LIN {X 0,Y 395.833,Z 526.81,A -85,B 0,C 180,E1 10637.81,E2 10637.81} C_VEL
LIN {X 0,Y 395.52,Z 526.81,A -85,B 0,C 180,E1 10644.894,E2 10644.894} C_VEL
LIN {X 0,Y 395.41,Z 526.81,A -85,B 0,C 180,E1 10649.844,E2 10649.844} C_VEL
LIN {X 0,Y 395.216,Z 526.81,A -85,B 0,C 180,E1 10656.446,E2 10656.446} C_VEL
LIN {X 0,Y 395.064,Z 526.81,A -85,B 0,C 180,E1 10663.606,E2 10663.606} C_VEL
LIN {X 0,Y 395.094,Z 526.81,A -85,B 0,C 180,E1 10670.021,E2 10670.021} C_VEL
LIN {X 0,Y 395.236,Z 526.81,A -85,B 0,C 180,E1 10677.573,E2 10677.573} C_VEL
LIN {X 0,Y 395.461,Z 526.81,A -85,B 0,C 180,E1 10679.651,E2 10679.651} C_VEL
LIN {X 0,Y 410.092,Z 574.473,A -85,B 0,C 180,E1 10681.377,E2 10681.377} C_VEL
LIN {X 0,Y 408.745,Z 609.401,A -85,B 0,C 180,E1 10682.378,E2 10682.378} C_VEL
LIN {X 0,Y 406.158,Z 642.659,A -85,B 0,C 180,E1 10684.177,E2 10684.177} C_VEL
LIN {X 0,Y 403.313,Z 673.055,A -85,B 0,C 180,E1 10686.737,E2 10686.737} C_VEL
LIN {X 0,Y 400.568,Z 700.736,A -85,B 0,C 180,E1 10690.118,E2 10690.118} C_VEL
LIN {X 0,Y 398.689,Z 723.257,A -85,B 0,C 180,E1 10694.024,E2 10694.024} C_VEL
LIN {X 0,Y 397.841,Z 740.947,A -85,B 0,C 180,E1 10698.48,E2 10698.48} C_VEL
LIN {X 0,Y 397.641,Z 746.134,A -85,B 0,C 180,E1 10700.254,E2 10700.254} C_VEL
LIN {X 0,Y 395.186,Z 750.11,A -85,B 0,C 180,E1 10702.034,E2 10702.034} C_VEL
LIN {X 0,Y 390.021,Z 754.134,A -85,B 0,C 180,E1 10704.784,E2 10704.784} C_VEL
LIN {X 0,Y 389.948,Z 754.482,A -85,B 0,C 180,E1 10705.103,E2 10705.103} C_VEL
LIN {X 0,Y 390.043,Z 756.982,A -85,B 0,C 180,E1 10707.781,E2 10707.781} C_VEL
LIN {X 0,Y 390.037,Z 756.855,A -85,B 0,C 180,E1 10712.23,E2 10712.23} C_VEL
LIN {X 0,Y 389.934,Z 751.669,A -85,B 0,C 180,E1 10716.695,E2 10716.695} C_VEL
LIN {X 0,Y 389.895,Z 741.071,A -85,B 0,C 180,E1 10721.201,E2 10721.201} C_VEL
LIN {X 0,Y 390.787,Z 724.457,A -85,B 0,C 180,E1 10725.742,E2 10725.742} C_VEL
LIN {X 0,Y 392.693,Z 701.933,A -85,B 0,C 180,E1 10730.001,E2 10730.001} C_VEL
LIN {X 0,Y 395.677,Z 676.121,A -85,B 0,C 180,E1 10733.488,E2 10733.488} C_VEL
LIN {X 0,Y 399.365,Z 644.916,A -85,B 0,C 180,E1 10736.459,E2 10736.459} C_VEL
LIN {X 0,Y 402.863,Z 611.392,A -85,B 0,C 180,E1 10738.55,E2 10738.55} C_VEL
LIN {X 0,Y 405.252,Z 576.378,A -85,B 0,C 180,E1 10739.789,E2 10739.789} C_VEL
LIN {X 0,Y 399.916,Z 555.834,A -85,B 0,C 180,E1 10740.82,E2 10740.82} C_VEL
LIN {X 0,Y 389.16,Z 531.813,A -85,B 0,C 180,E1 10742.683,E2 10742.683} C_VEL
LIN {X 0,Y 387.296,Z 526.81,A -85,B 0,C 180,E1 10743.189,E2 10743.189} C_VEL
LIN {X 0,Y 387.265,Z 526.81,A -85,B 0,C 180,E1 10748.729,E2 10748.729} C_VEL
LIN {X 0,Y 387.23,Z 526.81,A -85,B 0,C 180,E1 10755.28,E2 10755.28} C_VEL
LIN {X 0,Y 387.272,Z 526.81,A -85,B 0,C 180,E1 10761.445,E2 10761.445} C_VEL
LIN {X 0,Y 387.353,Z 526.81,A -85,B 0,C 180,E1 10766.833,E2 10766.833} C_VEL
LIN {X 0,Y 387.496,Z 526.81,A -85,B 0,C 180,E1 10773.997,E2 10773.997} C_VEL
LIN {X 0,Y 387.667,Z 527.164,A -85,B 0,C 180,E1 10777.454,E2 10777.454} C_VEL
LIN {X 0,Y 397.662,Z 554.122,A -85,B 0,C 180,E1 10779.969,E2 10779.969} C_VEL
LIN {X 0,Y 400.192,Z 572.611,A -85,B 0,C 180,E1 10781.611,E2 10781.611} C_VEL
LIN {X 0,Y 397.581,Z 598.094,A -85,B 0,C 180,E1 10784.122,E2 10784.122} C_VEL
LIN {X 0,Y 395.193,Z 617.876,A -85,B 0,C 180,E1 10787.083,E2 10787.083} C_VEL
LIN {X 0,Y 393.153,Z 633.028,A -85,B 0,C 180,E1 10790.587,E2 10790.587} C_VEL
LIN {X 0,Y 391.819,Z 642.578,A -85,B 0,C 180,E1 10794.463,E2 10794.463} C_VEL
LIN {X 0,Y 391.065,Z 645.829,A -85,B 0,C 180,E1 10797.788,E2 10797.788} C_VEL
LIN {X 0,Y 390.664,Z 644.811,A -85,B 0,C 180,E1 10801.117,E2 10801.117} C_VEL
LIN {X 0,Y 390.812,Z 638.222,A -85,B 0,C 180,E1 10805.007,E2 10805.007} C_VEL
LIN {X 0,Y 391.409,Z 626.317,A -85,B 0,C 180,E1 10808.627,E2 10808.627} C_VEL
LIN {X 0,Y 392.534,Z 608.81,A -85,B 0,C 180,E1 10811.972,E2 10811.972} C_VEL
LIN {X 0,Y 393.989,Z 587.013,A -85,B 0,C 180,E1 10814.756,E2 10814.756} C_VEL
LIN {X 0,Y 395.236,Z 562.293,A -85,B 0,C 180,E1 10816.869,E2 10816.869} C_VEL
LIN {X 0,Y 389.321,Z 533.266,A -85,B 0,C 180,E1 10818.647,E2 10818.647} C_VEL
LIN {X 0,Y 388.01,Z 526.81,A -85,B 0,C 180,E1 10818.953,E2 10818.953} C_VEL
LIN {X 0,Y 387.53,Z 526.81,A -85,B 0,C 180,E1 10826.013,E2 10826.013} C_VEL
LIN {X 0,Y 387.291,Z 526.81,A -85,B 0,C 180,E1 10833.189,E2 10833.189} C_VEL
LIN {X 0,Y 387.238,Z 526.81,A -85,B 0,C 180,E1 10838.732,E2 10838.732} C_VEL
LIN {X 0,Y 387.183,Z 526.81,A -85,B 0,C 180,E1 10845.253,E2 10845.253} C_VEL
LIN {X 0,Y 387.29,Z 526.81,A -85,B 0,C 180,E1 10851.44,E2 10851.44} C_VEL
LIN {X 0,Y 387.348,Z 526.81,A -85,B 0,C 180,E1 10856.816,E2 10856.816} C_VEL
LIN {X 0,Y 387.543,Z 526.81,A -85,B 0,C 180,E1 10863.981,E2 10863.981} C_VEL
LIN {X 0,Y 387.824,Z 526.81,A -85,B 0,C 180,E1 10869.559,E2 10869.559} C_VEL
LIN {X 0,Y 387.949,Z 526.81,A -85,B 0,C 180,E1 10876.452,E2 10876.452} C_VEL
LIN {X 0,Y 388.374,Z 526.81,A -85,B 0,C 180,E1 10883.278,E2 10883.278} C_VEL
LIN {X 0,Y 388.755,Z 526.81,A -85,B 0,C 180,E1 10889.995,E2 10889.995} C_VEL
LIN {X 0,Y 388.368,Z 526.81,A -85,B 0,C 180,E1 10896.711,E2 10896.711} C_VEL
LIN {X 0,Y 388.065,Z 526.81,A -85,B 0,C 180,E1 10903.533,E2 10903.533} C_VEL
LIN {X 0,Y 387.816,Z 526.81,A -85,B 0,C 180,E1 10910.565,E2 10910.565} C_VEL
LIN {X 0,Y 387.507,Z 526.81,A -85,B 0,C 180,E1 10917.955,E2 10917.955} C_VEL
LIN {X 0,Y 387.3,Z 526.81,A -85,B 0,C 180,E1 10924.812,E2 10924.812} C_VEL
LIN {X 0,Y 387.148,Z 526.81,A -85,B 0,C 180,E1 10932.001,E2 10932.001} C_VEL
LIN {X 0,Y 387.205,Z 526.81,A -85,B 0,C 180,E1 10938.331,E2 10938.331} C_VEL
LIN {X 0,Y 387.318,Z 526.81,A -85,B 0,C 180,E1 10945.167,E2 10945.167} C_VEL
LIN {X 0,Y 387.523,Z 526.81,A -85,B 0,C 180,E1 10952.034,E2 10952.034} C_VEL
LIN {X 0,Y 387.831,Z 526.81,A -85,B 0,C 180,E1 10959.529,E2 10959.529} C_VEL
LIN {X 0,Y 387.974,Z 526.81,A -85,B 0,C 180,E1 10966.452,E2 10966.452} C_VEL
LIN {X 0,Y 388.422,Z 526.81,A -85,B 0,C 180,E1 10973.278,E2 10973.278} C_VEL
LIN {X 0,Y 388.722,Z 526.81,A -85,B 0,C 180,E1 10979.993,E2 10979.993} C_VEL
LIN {X 0,Y 388.356,Z 526.81,A -85,B 0,C 180,E1 10986.709,E2 10986.709} C_VEL
LIN {X 0,Y 388.004,Z 526.81,A -85,B 0,C 180,E1 10993.533,E2 10993.533} C_VEL
LIN {X 0,Y 387.766,Z 526.81,A -85,B 0,C 180,E1 11000.565,E2 11000.565} C_VEL
LIN {X 0,Y 387.519,Z 526.81,A -85,B 0,C 180,E1 11007.95,E2 11007.95} C_VEL
LIN {X 0,Y 387.354,Z 526.81,A -85,B 0,C 180,E1 11014.841,E2 11014.841} C_VEL
LIN {X 0,Y 387.099,Z 526.81,A -85,B 0,C 180,E1 11022.007,E2 11022.007} C_VEL
LIN {X 0,Y 387.065,Z 526.81,A -85,B 0,C 180,E1 11028.326,E2 11028.326} C_VEL
LIN {X 0,Y 387.244,Z 526.81,A -85,B 0,C 180,E1 11035.176,E2 11035.176} C_VEL
LIN {X 0,Y 387.526,Z 527.326,A -85,B 0,C 180,E1 11039.247,E2 11039.247} C_VEL
LIN {X 0,Y 402.597,Z 575.135,A -85,B 0,C 180,E1 11041.032,E2 11041.032} C_VEL
LIN {X 0,Y 401.08,Z 610.921,A -85,B 0,C 180,E1 11042.117,E2 11042.117} C_VEL
LIN {X 0,Y 398.473,Z 643.198,A -85,B 0,C 180,E1 11043.944,E2 11043.944} C_VEL
LIN {X 0,Y 395.477,Z 673.867,A -85,B 0,C 180,E1 11046.625,E2 11046.625} C_VEL
LIN {X 0,Y 392.717,Z 700.654,A -85,B 0,C 180,E1 11050.008,E2 11050.008} C_VEL
LIN {X 0,Y 390.815,Z 722.905,A -85,B 0,C 180,E1 11053.982,E2 11053.982} C_VEL
LIN {X 0,Y 389.989,Z 739.481,A -85,B 0,C 180,E1 11058.245,E2 11058.245} C_VEL
LIN {X 0,Y 389.898,Z 750.617,A -85,B 0,C 180,E1 11062.621,E2 11062.621} C_VEL
LIN {X 0,Y 389.948,Z 754.482,A -85,B 0,C 180,E1 11065.103,E2 11065.103} C_VEL
LIN {X 0,Y 387.658,Z 756.165,A -85,B 0,C 180,E1 11066.987,E2 11066.987} C_VEL
LIN {X 0,Y 382.341,Z 756.336,A -85,B 0,C 180,E1 11070.182,E2 11070.182} C_VEL
LIN {X 0,Y 382.162,Z 753.806,A -85,B 0,C 180,E1 11074.55,E2 11074.55} C_VEL
LIN {X 0,Y 381.944,Z 745.92,A -85,B 0,C 180,E1 11079.129,E2 11079.129} C_VEL
LIN {X 0,Y 382.319,Z 732.498,A -85,B 0,C 180,E1 11083.751,E2 11083.751} C_VEL
LIN {X 0,Y 383.876,Z 712.313,A -85,B 0,C 180,E1 11088.399,E2 11088.399} C_VEL
LIN {X 0,Y 386.838,Z 687.296,A -85,B 0,C 180,E1 11092.439,E2 11092.439} C_VEL
LIN {X 0,Y 390.458,Z 658.719,A -85,B 0,C 180,E1 11095.716,E2 11095.716} C_VEL
LIN {X 0,Y 394.404,Z 626.331,A -85,B 0,C 180,E1 11098.253,E2 11098.253} C_VEL
LIN {X 0,Y 397.556,Z 592.247,A -85,B 0,C 180,E1 11099.916,E2 11099.916} C_VEL
LIN {X 0,Y 398.025,Z 574.069,A -85,B 0,C 180,E1 11100.508,E2 11100.508} C_VEL
LIN {X 0,Y 390.505,Z 550.725,A -85,B 0,C 180,E1 11101.947,E2 11101.947} C_VEL
LIN {X 0,Y 379.376,Z 526.81,A -85,B 0,C 180,E1 11104.174,E2 11104.174} C_VEL
LIN {X 0,Y 379.266,Z 526.81,A -85,B 0,C 180,E1 11110.682,E2 11110.682} C_VEL
LIN {X 0,Y 379.263,Z 526.81,A -85,B 0,C 180,E1 11117.273,E2 11117.273} C_VEL
LIN {X 0,Y 379.297,Z 526.81,A -85,B 0,C 180,E1 11123.229,E2 11123.229} C_VEL
LIN {X 0,Y 379.446,Z 526.81,A -85,B 0,C 180,E1 11128.763,E2 11128.763} C_VEL
LIN {X 0,Y 379.632,Z 526.81,A -85,B 0,C 180,E1 11136.364,E2 11136.364} C_VEL
LIN {X 0,Y 390.489,Z 554.777,A -85,B 0,C 180,E1 11139.28,E2 11139.28} C_VEL
LIN {X 0,Y 393.345,Z 573.867,A -85,B 0,C 180,E1 11141.074,E2 11141.074} C_VEL
LIN {X 0,Y 390.46,Z 599.555,A -85,B 0,C 180,E1 11143.68,E2 11143.68} C_VEL
LIN {X 0,Y 387.805,Z 619.699,A -85,B 0,C 180,E1 11146.776,E2 11146.776} C_VEL
LIN {X 0,Y 385.589,Z 634.811,A -85,B 0,C 180,E1 11150.401,E2 11150.401} C_VEL
LIN {X 0,Y 384.111,Z 644.058,A -85,B 0,C 180,E1 11154.352,E2 11154.352} C_VEL
LIN {X 0,Y 383.311,Z 647.144,A -85,B 0,C 180,E1 11157.743,E2 11157.743} C_VEL
LIN {X 0,Y 382.849,Z 645.949,A -85,B 0,C 180,E1 11161.14,E2 11161.14} C_VEL
LIN {X 0,Y 383.023,Z 639.115,A -85,B 0,C 180,E1 11165.109,E2 11165.109} C_VEL
LIN {X 0,Y 383.623,Z 626.948,A -85,B 0,C 180,E1 11168.804,E2 11168.804} C_VEL
LIN {X 0,Y 384.818,Z 609.109,A -85,B 0,C 180,E1 11172.216,E2 11172.216} C_VEL
LIN {X 0,Y 386.298,Z 586.882,A -85,B 0,C 180,E1 11175.056,E2 11175.056} C_VEL
LIN {X 0,Y 387.223,Z 561.791,A -85,B 0,C 180,E1 11177.213,E2 11177.213} C_VEL
LIN {X 0,Y 381.165,Z 532.299,A -85,B 0,C 180,E1 11179.02,E2 11179.02} C_VEL
LIN {X 0,Y 380.043,Z 526.81,A -85,B 0,C 180,E1 11179.299,E2 11179.299} C_VEL
LIN {X 0,Y 379.646,Z 526.81,A -85,B 0,C 180,E1 11186.027,E2 11186.027} C_VEL
LIN {X 0,Y 379.396,Z 526.81,A -85,B 0,C 180,E1 11193.055,E2 11193.055} C_VEL
LIN {X 0,Y 379.195,Z 526.81,A -85,B 0,C 180,E1 11200.647,E2 11200.647} C_VEL
LIN {X 0,Y 379.23,Z 526.81,A -85,B 0,C 180,E1 11207.249,E2 11207.249} C_VEL
LIN {X 0,Y 379.307,Z 526.81,A -85,B 0,C 180,E1 11213.213,E2 11213.213} C_VEL
LIN {X 0,Y 379.447,Z 526.81,A -85,B 0,C 180,E1 11218.747,E2 11218.747} C_VEL
LIN {X 0,Y 379.66,Z 526.81,A -85,B 0,C 180,E1 11223.975,E2 11223.975} C_VEL
LIN {X 0,Y 379.934,Z 526.81,A -85,B 0,C 180,E1 11231.404,E2 11231.404} C_VEL
LIN {X 0,Y 380.094,Z 526.81,A -85,B 0,C 180,E1 11238.506,E2 11238.506} C_VEL
LIN {X 0,Y 380.536,Z 526.81,A -85,B 0,C 180,E1 11245.43,E2 11245.43} C_VEL
LIN {X 0,Y 380.853,Z 526.81,A -85,B 0,C 180,E1 11249.995,E2 11249.995} C_VEL
LIN {X 0,Y 380.457,Z 526.81,A -85,B 0,C 180,E1 11256.851,E2 11256.851} C_VEL
LIN {X 0,Y 380.121,Z 526.81,A -85,B 0,C 180,E1 11263.821,E2 11263.821} C_VEL
LIN {X 0,Y 379.834,Z 526.81,A -85,B 0,C 180,E1 11271.018,E2 11271.018} C_VEL
LIN {X 0,Y 379.524,Z 526.81,A -85,B 0,C 180,E1 11278.629,E2 11278.629} C_VEL
LIN {X 0,Y 379.366,Z 526.81,A -85,B 0,C 180,E1 11283.963,E2 11283.963} C_VEL
LIN {X 0,Y 379.166,Z 526.81,A -85,B 0,C 180,E1 11290.643,E2 11290.643} C_VEL
LIN {X 0,Y 379.233,Z 526.81,A -85,B 0,C 180,E1 11297.25,E2 11297.25} C_VEL
LIN {X 0,Y 379.283,Z 526.81,A -85,B 0,C 180,E1 11303.21,E2 11303.21} C_VEL
LIN {X 0,Y 379.42,Z 526.81,A -85,B 0,C 180,E1 11308.744,E2 11308.744} C_VEL
LIN {X 0,Y 379.709,Z 526.81,A -85,B 0,C 180,E1 11316.494,E2 11316.494} C_VEL
LIN {X 0,Y 379.995,Z 526.81,A -85,B 0,C 180,E1 11323.798,E2 11323.798} C_VEL
LIN {X 0,Y 380.291,Z 526.81,A -85,B 0,C 180,E1 11331.518,E2 11331.518} C_VEL
LIN {X 0,Y 380.78,Z 526.81,A -85,B 0,C 180,E1 11337.714,E2 11337.714} C_VEL
LIN {X 0,Y 380.594,Z 526.81,A -85,B 0,C 180,E1 11344.556,E2 11344.556} C_VEL
LIN {X 0,Y 380.149,Z 526.81,A -85,B 0,C 180,E1 11351.479,E2 11351.479} C_VEL
LIN {X 0,Y 379.929,Z 526.81,A -85,B 0,C 180,E1 11358.583,E2 11358.583} C_VEL
LIN {X 0,Y 379.626,Z 526.81,A -85,B 0,C 180,E1 11366.013,E2 11366.013} C_VEL
LIN {X 0,Y 379.446,Z 526.81,A -85,B 0,C 180,E1 11373.951,E2 11373.951} C_VEL
LIN {X 0,Y 379.154,Z 526.81,A -85,B 0,C 180,E1 11380.657,E2 11380.657} C_VEL
LIN {X 0,Y 379.074,Z 526.81,A -85,B 0,C 180,E1 11387.242,E2 11387.242} C_VEL
LIN {X 0,Y 379.181,Z 526.81,A -85,B 0,C 180,E1 11393.212,E2 11393.212} C_VEL
LIN {X 0,Y 379.575,Z 526.81,A -85,B 0,C 180,E1 11398.771,E2 11398.771} C_VEL
LIN {X 0,Y 395.009,Z 576.235,A -85,B 0,C 180,E1 11400.686,E2 11400.686} C_VEL
LIN {X 0,Y 393.505,Z 611.185,A -85,B 0,C 180,E1 11401.801,E2 11401.801} C_VEL
LIN {X 0,Y 390.686,Z 644.506,A -85,B 0,C 180,E1 11403.765,E2 11403.765} C_VEL
LIN {X 0,Y 387.684,Z 673.91,A -85,B 0,C 180,E1 11406.434,E2 11406.434} C_VEL
LIN {X 0,Y 384.8,Z 701.173,A -85,B 0,C 180,E1 11410.003,E2 11410.003} C_VEL
LIN {X 0,Y 382.933,Z 722.47,A -85,B 0,C 180,E1 11413.938,E2 11413.938} C_VEL
LIN {X 0,Y 382.09,Z 739.805,A -85,B 0,C 180,E1 11418.578,E2 11418.578} C_VEL
LIN {X 0,Y 382.104,Z 750.549,A -85,B 0,C 180,E1 11423.178,E2 11423.178} C_VEL
LIN {X 0,Y 382.217,Z 755.777,A -85,B 0,C 180,E1 11427.735,E2 11427.735} C_VEL
LIN {X 0,Y 382.341,Z 756.336,A -85,B 0,C 180,E1 11430.182,E2 11430.182} C_VEL
LIN {X 0,Y 379.656,Z 755.445,A -85,B 0,C 180,E1 11432.103,E2 11432.103} C_VEL
LIN {X 0,Y 374.266,Z 751.83,A -85,B 0,C 180,E1 11435.303,E2 11435.303} C_VEL
LIN {X 0,Y 374.054,Z 743.465,A -85,B 0,C 180,E1 11439.911,E2 11439.911} C_VEL
LIN {X 0,Y 374.633,Z 729.252,A -85,B 0,C 180,E1 11444.637,E2 11444.637} C_VEL
LIN {X 0,Y 376.399,Z 709.724,A -85,B 0,C 180,E1 11449.092,E2 11449.092} C_VEL
LIN {X 0,Y 379.627,Z 684.333,A -85,B 0,C 180,E1 11453.2,E2 11453.2} C_VEL
LIN {X 0,Y 383.506,Z 655.208,A -85,B 0,C 180,E1 11456.533,E2 11456.533} C_VEL
LIN {X 0,Y 387.98,Z 621.858,A -85,B 0,C 180,E1 11459.087,E2 11459.087} C_VEL
LIN {X 0,Y 391.317,Z 587.429,A -85,B 0,C 180,E1 11460.699,E2 11460.699} C_VEL
LIN {X 0,Y 391.301,Z 575.135,A -85,B 0,C 180,E1 11461.139,E2 11461.139} C_VEL
LIN {X 0,Y 383.806,Z 552.489,A -85,B 0,C 180,E1 11462.667,E2 11462.667} C_VEL
LIN {X 0,Y 372.915,Z 531.315,A -85,B 0,C 180,E1 11464.919,E2 11464.919} C_VEL
LIN {X 0,Y 371.481,Z 526.81,A -85,B 0,C 180,E1 11465.414,E2 11465.414} C_VEL
LIN {X 0,Y 371.381,Z 526.81,A -85,B 0,C 180,E1 11472.805,E2 11472.805} C_VEL
LIN {X 0,Y 371.368,Z 526.81,A -85,B 0,C 180,E1 11479.295,E2 11479.295} C_VEL
LIN {X 0,Y 371.392,Z 526.81,A -85,B 0,C 180,E1 11485.209,E2 11485.209} C_VEL
LIN {X 0,Y 371.555,Z 526.81,A -85,B 0,C 180,E1 11490.735,E2 11490.735} C_VEL
LIN {X 0,Y 371.721,Z 527.201,A -85,B 0,C 180,E1 11495.261,E2 11495.261} C_VEL
LIN {X 0,Y 383.001,Z 554.104,A -85,B 0,C 180,E1 11498.393,E2 11498.393} C_VEL
LIN {X 0,Y 386.609,Z 574.886,A -85,B 0,C 180,E1 11500.487,E2 11500.487} C_VEL
LIN {X 0,Y 383.394,Z 601.235,A -85,B 0,C 180,E1 11503.223,E2 11503.223} C_VEL
LIN {X 0,Y 380.485,Z 621.376,A -85,B 0,C 180,E1 11506.414,E2 11506.414} C_VEL
LIN {X 0,Y 378.267,Z 635.03,A -85,B 0,C 180,E1 11509.704,E2 11509.704} C_VEL
LIN {X 0,Y 376.74,Z 643.717,A -85,B 0,C 180,E1 11513.083,E2 11513.083} C_VEL
LIN {X 0,Y 376.091,Z 647.017,A -85,B 0,C 180,E1 11515.389,E2 11515.389} C_VEL
LIN {X 0,Y 375.545,Z 648.445,A -85,B 0,C 180,E1 11517.697,E2 11517.697} C_VEL
LIN {X 0,Y 375.051,Z 647.071,A -85,B 0,C 180,E1 11521.164,E2 11521.164} C_VEL
LIN {X 0,Y 375.204,Z 639.959,A -85,B 0,C 180,E1 11525.216,E2 11525.216} C_VEL
LIN {X 0,Y 375.844,Z 627.545,A -85,B 0,C 180,E1 11528.984,E2 11528.984} C_VEL
LIN {X 0,Y 377.082,Z 609.407,A -85,B 0,C 180,E1 11532.47,E2 11532.47} C_VEL
LIN {X 0,Y 378.751,Z 585.397,A -85,B 0,C 180,E1 11535.512,E2 11535.512} C_VEL
LIN {X 0,Y 379.458,Z 562.632,A -85,B 0,C 180,E1 11537.466,E2 11537.466} C_VEL
LIN {X 0,Y 373.527,Z 533.469,A -85,B 0,C 180,E1 11539.309,E2 11539.309} C_VEL
LIN {X 0,Y 372.132,Z 526.81,A -85,B 0,C 180,E1 11539.606,E2 11539.606} C_VEL
LIN {X 0,Y 371.66,Z 526.81,A -85,B 0,C 180,E1 11546.63,E2 11546.63} C_VEL
LIN {X 0,Y 371.482,Z 526.81,A -85,B 0,C 180,E1 11552.002,E2 11552.002} C_VEL
LIN {X 0,Y 371.281,Z 526.81,A -85,B 0,C 180,E1 11559.203,E2 11559.203} C_VEL
LIN {X 0,Y 371.309,Z 526.81,A -85,B 0,C 180,E1 11566.108,E2 11566.108} C_VEL
LIN {X 0,Y 371.306,Z 526.81,A -85,B 0,C 180,E1 11572.284,E2 11572.284} C_VEL
LIN {X 0,Y 371.539,Z 526.81,A -85,B 0,C 180,E1 11578.855,E2 11578.855} C_VEL
LIN {X 0,Y 371.751,Z 526.81,A -85,B 0,C 180,E1 11585.96,E2 11585.96} C_VEL
LIN {X 0,Y 371.967,Z 526.81,A -85,B 0,C 180,E1 11590.99,E2 11590.99} C_VEL
LIN {X 0,Y 372.154,Z 526.81,A -85,B 0,C 180,E1 11598.257,E2 11598.257} C_VEL
LIN {X 0,Y 372.623,Z 526.81,A -85,B 0,C 180,E1 11605.333,E2 11605.333} C_VEL
LIN {X 0,Y 372.951,Z 526.81,A -85,B 0,C 180,E1 11609.994,E2 11609.994} C_VEL
LIN {X 0,Y 372.53,Z 526.81,A -85,B 0,C 180,E1 11616.998,E2 11616.998} C_VEL
LIN {X 0,Y 372.178,Z 526.81,A -85,B 0,C 180,E1 11624.122,E2 11624.122} C_VEL
LIN {X 0,Y 371.857,Z 526.81,A -85,B 0,C 180,E1 11631.491,E2 11631.491} C_VEL
LIN {X 0,Y 371.632,Z 526.81,A -85,B 0,C 180,E1 11636.619,E2 11636.619} C_VEL
LIN {X 0,Y 371.484,Z 526.81,A -85,B 0,C 180,E1 11641.988,E2 11641.988} C_VEL
LIN {X 0,Y 371.252,Z 526.81,A -85,B 0,C 180,E1 11649.199,E2 11649.199} C_VEL
LIN {X 0,Y 371.291,Z 526.81,A -85,B 0,C 180,E1 11656.106,E2 11656.106} C_VEL
LIN {X 0,Y 371.286,Z 526.81,A -85,B 0,C 180,E1 11662.282,E2 11662.282} C_VEL
LIN {X 0,Y 371.509,Z 526.81,A -85,B 0,C 180,E1 11668.842,E2 11668.842} C_VEL
LIN {X 0,Y 371.732,Z 526.81,A -85,B 0,C 180,E1 11675.958,E2 11675.958} C_VEL
LIN {X 0,Y 371.991,Z 526.81,A -85,B 0,C 180,E1 11680.991,E2 11680.991} C_VEL
LIN {X 0,Y 372.17,Z 526.81,A -85,B 0,C 180,E1 11688.257,E2 11688.257} C_VEL
LIN {X 0,Y 372.61,Z 526.81,A -85,B 0,C 180,E1 11695.332,E2 11695.332} C_VEL
LIN {X 0,Y 372.837,Z 526.81,A -85,B 0,C 180,E1 11702.32,E2 11702.32} C_VEL
LIN {X 0,Y 372.351,Z 526.81,A -85,B 0,C 180,E1 11709.353,E2 11709.353} C_VEL
LIN {X 0,Y 372.084,Z 526.81,A -85,B 0,C 180,E1 11716.541,E2 11716.541} C_VEL
LIN {X 0,Y 371.814,Z 526.81,A -85,B 0,C 180,E1 11721.49,E2 11721.49} C_VEL
LIN {X 0,Y 371.654,Z 526.81,A -85,B 0,C 180,E1 11726.614,E2 11726.614} C_VEL
LIN {X 0,Y 371.508,Z 526.81,A -85,B 0,C 180,E1 11731.982,E2 11731.982} C_VEL
LIN {X 0,Y 371.276,Z 526.81,A -85,B 0,C 180,E1 11739.22,E2 11739.22} C_VEL
LIN {X 0,Y 371.162,Z 526.81,A -85,B 0,C 180,E1 11746.102,E2 11746.102} C_VEL
LIN {X 0,Y 371.173,Z 526.81,A -85,B 0,C 180,E1 11752.282,E2 11752.282} C_VEL
LIN {X 0,Y 371.62,Z 526.81,A -85,B 0,C 180,E1 11758.357,E2 11758.357} C_VEL
LIN {X 0,Y 387.541,Z 577.763,A -85,B 0,C 180,E1 11760.356,E2 11760.356} C_VEL
LIN {X 0,Y 385.852,Z 612.406,A -85,B 0,C 180,E1 11761.526,E2 11761.526} C_VEL
LIN {X 0,Y 382.941,Z 645.126,A -85,B 0,C 180,E1 11763.54,E2 11763.54} C_VEL
LIN {X 0,Y 379.793,Z 675.058,A -85,B 0,C 180,E1 11766.372,E2 11766.372} C_VEL
LIN {X 0,Y 376.896,Z 701.419,A -85,B 0,C 180,E1 11769.962,E2 11769.962} C_VEL
LIN {X 0,Y 374.984,Z 723.271,A -85,B 0,C 180,E1 11774.191,E2 11774.191} C_VEL
LIN {X 0,Y 374.23,Z 739.943,A -85,B 0,C 180,E1 11778.926,E2 11778.926} C_VEL
LIN {X 0,Y 374.273,Z 749.206,A -85,B 0,C 180,E1 11783.035,E2 11783.035} C_VEL
LIN {X 0,Y 374.409,Z 754.542,A -85,B 0,C 180,E1 11787.688,E2 11787.688} C_VEL
LIN {X 0,Y 374.401,Z 754.554,A -85,B 0,C 180,E1 11792.323,E2 11792.323} C_VEL
LIN {X 0,Y 374.266,Z 751.83,A -85,B 0,C 180,E1 11795.303,E2 11795.303} C_VEL
LIN {X 0,Y 371.643,Z 748.735,A -85,B 0,C 180,E1 11797.222,E2 11797.222} C_VEL
LIN {X 0,Y 366.27,Z 742.551,A -85,B 0,C 180,E1 11800.045,E2 11800.045} C_VEL
LIN {X 0,Y 366.196,Z 741.78,A -85,B 0,C 180,E1 11800.37,E2 11800.37} C_VEL
LIN {X 0,Y 366.888,Z 727.12,A -85,B 0,C 180,E1 11805.259,E2 11805.259} C_VEL
LIN {X 0,Y 368.886,Z 707.269,A -85,B 0,C 180,E1 11809.798,E2 11809.798} C_VEL
LIN {X 0,Y 372.458,Z 681.39,A -85,B 0,C 180,E1 11813.992,E2 11813.992} C_VEL
LIN {X 0,Y 376.746,Z 652.603,A -85,B 0,C 180,E1 11817.283,E2 11817.283} C_VEL
LIN {X 0,Y 381.426,Z 619.331,A -85,B 0,C 180,E1 11819.836,E2 11819.836} C_VEL
LIN {X 0,Y 384.969,Z 584.686,A -85,B 0,C 180,E1 11821.451,E2 11821.451} C_VEL
LIN {X 0,Y 384.345,Z 574.581,A -85,B 0,C 180,E1 11821.901,E2 11821.901} C_VEL
LIN {X 0,Y 375.655,Z 550.859,A -85,B 0,C 180,E1 11823.775,E2 11823.775} C_VEL
LIN {X 0,Y 365.632,Z 532.243,A -85,B 0,C 180,E1 11826.087,E2 11826.087} C_VEL
LIN {X 0,Y 363.398,Z 526.81,A -85,B 0,C 180,E1 11826.887,E2 11826.887} C_VEL
LIN {X 0,Y 363.432,Z 526.81,A -85,B 0,C 180,E1 11831.81,E2 11831.81} C_VEL
LIN {X 0,Y 363.426,Z 526.81,A -85,B 0,C 180,E1 11838.59,E2 11838.59} C_VEL
LIN {X 0,Y 363.414,Z 526.81,A -85,B 0,C 180,E1 11844.33,E2 11844.33} C_VEL
LIN {X 0,Y 363.642,Z 526.81,A -85,B 0,C 180,E1 11850.981,E2 11850.981} C_VEL
LIN {X 0,Y 363.783,Z 527.355,A -85,B 0,C 180,E1 11853.92,E2 11853.92} C_VEL
LIN {X 0,Y 375.307,Z 552.971,A -85,B 0,C 180,E1 11857.347,E2 11857.347} C_VEL
LIN {X 0,Y 379.906,Z 574.8,A -85,B 0,C 180,E1 11859.747,E2 11859.747} C_VEL
LIN {X 0,Y 376.71,Z 600.818,A -85,B 0,C 180,E1 11862.464,E2 11862.464} C_VEL
LIN {X 0,Y 373.562,Z 621.065,A -85,B 0,C 180,E1 11865.634,E2 11865.634} C_VEL
LIN {X 0,Y 370.797,Z 636.696,A -85,B 0,C 180,E1 11869.42,E2 11869.42} C_VEL
LIN {X 0,Y 369.06,Z 645.324,A -85,B 0,C 180,E1 11872.938,E2 11872.938} C_VEL
LIN {X 0,Y 368.376,Z 648.499,A -85,B 0,C 180,E1 11875.292,E2 11875.292} C_VEL
LIN {X 0,Y 367.792,Z 649.76,A -85,B 0,C 180,E1 11877.648,E2 11877.648} C_VEL
LIN {X 0,Y 367.23,Z 648.172,A -85,B 0,C 180,E1 11881.188,E2 11881.188} C_VEL
LIN {X 0,Y 367.388,Z 640.792,A -85,B 0,C 180,E1 11885.328,E2 11885.328} C_VEL
LIN {X 0,Y 368.049,Z 628.342,A -85,B 0,C 180,E1 11889.105,E2 11889.105} C_VEL
LIN {X 0,Y 369.339,Z 609.56,A -85,B 0,C 180,E1 11892.736,E2 11892.736} C_VEL
LIN {X 0,Y 371,Z 586.524,A -85,B 0,C 180,E1 11895.693,E2 11895.693} C_VEL
LIN {X 0,Y 371.667,Z 563.202,A -85,B 0,C 180,E1 11897.744,E2 11897.744} C_VEL
LIN {X 0,Y 365.717,Z 534.003,A -85,B 0,C 180,E1 11899.616,E2 11899.616} C_VEL
LIN {X 0,Y 364.164,Z 526.81,A -85,B 0,C 180,E1 11899.983,E2 11899.983} C_VEL
LIN {X 0,Y 363.66,Z 526.81,A -85,B 0,C 180,E1 11907.263,E2 11907.263} C_VEL
LIN {X 0,Y 363.395,Z 526.81,A -85,B 0,C 180,E1 11913.552,E2 11913.552} C_VEL
LIN {X 0,Y 363.38,Z 526.81,A -85,B 0,C 180,E1 11918.689,E2 11918.689} C_VEL
LIN {X 0,Y 363.354,Z 526.81,A -85,B 0,C 180,E1 11925.11,E2 11925.11} C_VEL
LIN {X 0,Y 363.419,Z 526.81,A -85,B 0,C 180,E1 11932.341,E2 11932.341} C_VEL
LIN {X 0,Y 363.647,Z 526.81,A -85,B 0,C 180,E1 11940.018,E2 11940.018} C_VEL
LIN {X 0,Y 363.883,Z 526.81,A -85,B 0,C 180,E1 11948.002,E2 11948.002} C_VEL
LIN {X 0,Y 364.138,Z 526.81,A -85,B 0,C 180,E1 11955.548,E2 11955.548} C_VEL
LIN {X 0,Y 364.606,Z 526.81,A -85,B 0,C 180,E1 11962.838,E2 11962.838} C_VEL
LIN {X 0,Y 365.049,Z 526.81,A -85,B 0,C 180,E1 11969.994,E2 11969.994} C_VEL
LIN {X 0,Y 364.608,Z 526.81,A -85,B 0,C 180,E1 11977.151,E2 11977.151} C_VEL
LIN {X 0,Y 364.234,Z 526.81,A -85,B 0,C 180,E1 11984.437,E2 11984.437} C_VEL
LIN {X 0,Y 363.872,Z 526.81,A -85,B 0,C 180,E1 11991.987,E2 11991.987} C_VEL
LIN {X 0,Y 363.611,Z 526.81,A -85,B 0,C 180,E1 11999.972,E2 11999.972} C_VEL
LIN {X 0,Y 363.355,Z 526.81,A -85,B 0,C 180,E1 12007.646,E2 12007.646} C_VEL
LIN {X 0,Y 363.324,Z 526.81,A -85,B 0,C 180,E1 12015.1,E2 12015.1} C_VEL
LIN {X 0,Y 363.396,Z 526.81,A -85,B 0,C 180,E1 12022.328,E2 12022.328} C_VEL
LIN {X 0,Y 363.612,Z 526.81,A -85,B 0,C 180,E1 12030.015,E2 12030.015} C_VEL
LIN {X 0,Y 363.875,Z 526.81,A -85,B 0,C 180,E1 12038.001,E2 12038.001} C_VEL
LIN {X 0,Y 364.16,Z 526.81,A -85,B 0,C 180,E1 12043.073,E2 12043.073} C_VEL
LIN {X 0,Y 364.406,Z 526.81,A -85,B 0,C 180,E1 12050.426,E2 12050.426} C_VEL
LIN {X 0,Y 364.948,Z 526.81,A -85,B 0,C 180,E1 12057.615,E2 12057.615} C_VEL
LIN {X 0,Y 364.772,Z 526.81,A -85,B 0,C 180,E1 12064.754,E2 12064.754} C_VEL
LIN {X 0,Y 364.291,Z 526.81,A -85,B 0,C 180,E1 12071.986,E2 12071.986} C_VEL
LIN {X 0,Y 364.032,Z 526.81,A -85,B 0,C 180,E1 12079.426,E2 12079.426} C_VEL
LIN {X 0,Y 363.745,Z 526.81,A -85,B 0,C 180,E1 12084.588,E2 12084.588} C_VEL
LIN {X 0,Y 363.63,Z 526.81,A -85,B 0,C 180,E1 12089.967,E2 12089.967} C_VEL
LIN {X 0,Y 363.401,Z 526.81,A -85,B 0,C 180,E1 12097.673,E2 12097.673} C_VEL
LIN {X 0,Y 363.226,Z 526.81,A -85,B 0,C 180,E1 12105.11,E2 12105.11} C_VEL
LIN {X 0,Y 363.288,Z 526.81,A -85,B 0,C 180,E1 12112.344,E2 12112.344} C_VEL
LIN {X 0,Y 363.658,Z 526.81,A -85,B 0,C 180,E1 12117.896,E2 12117.896} C_VEL
LIN {X 0,Y 380.034,Z 580.929,A -85,B 0,C 180,E1 12120.069,E2 12120.069} C_VEL
LIN {X 0,Y 378.002,Z 615.23,A -85,B 0,C 180,E1 12121.345,E2 12121.345} C_VEL
LIN {X 0,Y 374.921,Z 648.185,A -85,B 0,C 180,E1 12123.527,E2 12123.527} C_VEL
LIN {X 0,Y 371.71,Z 677.866,A -85,B 0,C 180,E1 12126.527,E2 12126.527} C_VEL
LIN {X 0,Y 368.798,Z 703.313,A -85,B 0,C 180,E1 12130.208,E2 12130.208} C_VEL
LIN {X 0,Y 367.031,Z 723.995,A -85,B 0,C 180,E1 12134.452,E2 12134.452} C_VEL
LIN {X 0,Y 366.354,Z 740.033,A -85,B 0,C 180,E1 12139.288,E2 12139.288} C_VEL
LIN {X 0,Y 366.497,Z 749.722,A -85,B 0,C 180,E1 12144.078,E2 12144.078} C_VEL
LIN {X 0,Y 366.589,Z 753.283,A -85,B 0,C 180,E1 12147.639,E2 12147.639} C_VEL
LIN {X 0,Y 366.752,Z 753.995,A -85,B 0,C 180,E1 12150.006,E2 12150.006} C_VEL
LIN {X 0,Y 366.487,Z 751.512,A -85,B 0,C 180,E1 12154.745,E2 12154.745} C_VEL
LIN {X 0,Y 366.202,Z 743.708,A -85,B 0,C 180,E1 12159.525,E2 12159.525} C_VEL
LIN {X 0,Y 366.196,Z 741.78,A -85,B 0,C 180,E1 12160.37,E2 12160.37} C_VEL
LIN {X 0,Y 363.782,Z 736.874,A -85,B 0,C 180,E1 12162.248,E2 12162.248} C_VEL
LIN {X 0,Y 358.975,Z 728.295,A -85,B 0,C 180,E1 12164.986,E2 12164.986} C_VEL
LIN {X 0,Y 359,Z 727.21,A -85,B 0,C 180,E1 12165.292,E2 12165.292} C_VEL
LIN {X 0,Y 361.228,Z 706.421,A -85,B 0,C 180,E1 12170.236,E2 12170.236} C_VEL
LIN {X 0,Y 365.12,Z 680.801,A -85,B 0,C 180,E1 12174.505,E2 12174.505} C_VEL
LIN {X 0,Y 369.858,Z 651.223,A -85,B 0,C 180,E1 12177.966,E2 12177.966} C_VEL
LIN {X 0,Y 374.774,Z 618.854,A -85,B 0,C 180,E1 12180.505,E2 12180.505} C_VEL
LIN {X 0,Y 378.6,Z 584.798,A -85,B 0,C 180,E1 12182.153,E2 12182.153} C_VEL
LIN {X 0,Y 377.63,Z 575.062,A -85,B 0,C 180,E1 12182.669,E2 12182.669} C_VEL
LIN {X 0,Y 368.951,Z 552.256,A -85,B 0,C 180,E1 12184.696,E2 12184.696} C_VEL
LIN {X 0,Y 358.486,Z 532.983,A -85,B 0,C 180,E1 12187.412,E2 12187.412} C_VEL
LIN {X 0,Y 355.579,Z 528.042,A -85,B 0,C 180,E1 12188.313,E2 12188.313} C_VEL
LIN {X 0,Y 355.508,Z 526.81,A -85,B 0,C 180,E1 12188.471,E2 12188.471} C_VEL
LIN {X 0,Y 355.373,Z 526.81,A -85,B 0,C 180,E1 12196.418,E2 12196.418} C_VEL
LIN {X 0,Y 355.498,Z 526.81,A -85,B 0,C 180,E1 12204.029,E2 12204.029} C_VEL
LIN {X 0,Y 355.734,Z 526.81,A -85,B 0,C 180,E1 12212.094,E2 12212.094} C_VEL
LIN {X 0,Y 358.567,Z 532.8,A -85,B 0,C 180,E1 12213.294,E2 12213.294} C_VEL
LIN {X 0,Y 368.62,Z 554.7,A -85,B 0,C 180,E1 12216.543,E2 12216.543} C_VEL
LIN {X 0,Y 373.146,Z 575.119,A -85,B 0,C 180,E1 12218.961,E2 12218.961} C_VEL
LIN {X 0,Y 369.959,Z 601.696,A -85,B 0,C 180,E1 12221.825,E2 12221.825} C_VEL
LIN {X 0,Y 366.521,Z 621.947,A -85,B 0,C 180,E1 12225.046,E2 12225.046} C_VEL
LIN {X 0,Y 363.616,Z 636.514,A -85,B 0,C 180,E1 12228.513,E2 12228.513} C_VEL
LIN {X 0,Y 361.42,Z 646.982,A -85,B 0,C 180,E1 12232.788,E2 12232.788} C_VEL
LIN {X 0,Y 360.672,Z 649.995,A -85,B 0,C 180,E1 12235.192,E2 12235.192} C_VEL
LIN {X 0,Y 360.041,Z 651.075,A -85,B 0,C 180,E1 12237.597,E2 12237.597} C_VEL
LIN {X 0,Y 359.413,Z 649.244,A -85,B 0,C 180,E1 12241.214,E2 12241.214} C_VEL
LIN {X 0,Y 359.562,Z 641.618,A -85,B 0,C 180,E1 12245.444,E2 12245.444} C_VEL
LIN {X 0,Y 360.26,Z 628.834,A -85,B 0,C 180,E1 12249.303,E2 12249.303} C_VEL
LIN {X 0,Y 361.611,Z 609.629,A -85,B 0,C 180,E1 12253.013,E2 12253.013} C_VEL
LIN {X 0,Y 363.301,Z 586.673,A -85,B 0,C 180,E1 12255.974,E2 12255.974} C_VEL
LIN {X 0,Y 364.091,Z 565.169,A -85,B 0,C 180,E1 12257.903,E2 12257.903} C_VEL
LIN {X 0,Y 357.99,Z 534.912,A -85,B 0,C 180,E1 12259.917,E2 12259.917} C_VEL
LIN {X 0,Y 356.207,Z 526.81,A -85,B 0,C 180,E1 12260.367,E2 12260.367} C_VEL
LIN {X 0,Y 355.729,Z 526.81,A -85,B 0,C 180,E1 12267.924,E2 12267.924} C_VEL
LIN {X 0,Y 355.463,Z 526.81,A -85,B 0,C 180,E1 12275.964,E2 12275.964} C_VEL
LIN {X 0,Y 355.329,Z 526.81,A -85,B 0,C 180,E1 12283.575,E2 12283.575} C_VEL
LIN {X 0,Y 355.422,Z 526.81,A -85,B 0,C 180,E1 12290.276,E2 12290.276} C_VEL
LIN {X 0,Y 355.537,Z 526.81,A -85,B 0,C 180,E1 12296.378,E2 12296.378} C_VEL
LIN {X 0,Y 355.763,Z 526.81,A -85,B 0,C 180,E1 12303.356,E2 12303.356} C_VEL
LIN {X 0,Y 356.064,Z 526.81,A -85,B 0,C 180,E1 12310.106,E2 12310.106} C_VEL
LIN {X 0,Y 356.333,Z 526.81,A -85,B 0,C 180,E1 12317.784,E2 12317.784} C_VEL
LIN {X 0,Y 356.814,Z 526.81,A -85,B 0,C 180,E1 12325.126,E2 12325.126} C_VEL
LIN {X 0,Y 357.161,Z 526.81,A -85,B 0,C 180,E1 12329.994,E2 12329.994} C_VEL
LIN {X 0,Y 356.676,Z 526.81,A -85,B 0,C 180,E1 12337.311,E2 12337.311} C_VEL
LIN {X 0,Y 356.286,Z 526.81,A -85,B 0,C 180,E1 12344.766,E2 12344.766} C_VEL
LIN {X 0,Y 355.915,Z 526.81,A -85,B 0,C 180,E1 12352.505,E2 12352.505} C_VEL
LIN {X 0,Y 355.709,Z 526.81,A -85,B 0,C 180,E1 12357.912,E2 12357.912} C_VEL
LIN {X 0,Y 355.455,Z 526.81,A -85,B 0,C 180,E1 12365.963,E2 12365.963} C_VEL
LIN {X 0,Y 355.298,Z 526.81,A -85,B 0,C 180,E1 12373.57,E2 12373.57} C_VEL
LIN {X 0,Y 355.407,Z 526.81,A -85,B 0,C 180,E1 12380.274,E2 12380.274} C_VEL
LIN {X 0,Y 355.508,Z 526.81,A -85,B 0,C 180,E1 12386.375,E2 12386.375} C_VEL
LIN {X 0,Y 355.745,Z 526.81,A -85,B 0,C 180,E1 12393.338,E2 12393.338} C_VEL
LIN {X 0,Y 356.079,Z 526.81,A -85,B 0,C 180,E1 12400.106,E2 12400.106} C_VEL
LIN {X 0,Y 356.343,Z 526.81,A -85,B 0,C 180,E1 12407.727,E2 12407.727} C_VEL
LIN {X 0,Y 356.826,Z 526.81,A -85,B 0,C 180,E1 12415.125,E2 12415.125} C_VEL
LIN {X 0,Y 357.128,Z 526.81,A -85,B 0,C 180,E1 12419.993,E2 12419.993} C_VEL
LIN {X 0,Y 356.664,Z 526.81,A -85,B 0,C 180,E1 12427.309,E2 12427.309} C_VEL
LIN {X 0,Y 356.233,Z 526.81,A -85,B 0,C 180,E1 12434.766,E2 12434.766} C_VEL
LIN {X 0,Y 355.891,Z 526.81,A -85,B 0,C 180,E1 12442.503,E2 12442.503} C_VEL
LIN {X 0,Y 355.738,Z 526.81,A -85,B 0,C 180,E1 12447.906,E2 12447.906} C_VEL
LIN {X 0,Y 355.56,Z 526.81,A -85,B 0,C 180,E1 12453.602,E2 12453.602} C_VEL
LIN {X 0,Y 355.348,Z 526.81,A -85,B 0,C 180,E1 12459.929,E2 12459.929} C_VEL
LIN {X 0,Y 355.213,Z 526.81,A -85,B 0,C 180,E1 12467.009,E2 12467.009} C_VEL
LIN {X 0,Y 355.392,Z 526.81,A -85,B 0,C 180,E1 12474.026,E2 12474.026} C_VEL
LIN {X 0,Y 355.644,Z 526.81,A -85,B 0,C 180,E1 12477.461,E2 12477.461} C_VEL
LIN {X 0,Y 372.477,Z 583.035,A -85,B 0,C 180,E1 12479.75,E2 12479.75} C_VEL
LIN {X 0,Y 370.279,Z 616.517,A -85,B 0,C 180,E1 12481.086,E2 12481.086} C_VEL
LIN {X 0,Y 367.095,Z 649.225,A -85,B 0,C 180,E1 12483.357,E2 12483.357} C_VEL
LIN {X 0,Y 363.771,Z 678.796,A -85,B 0,C 180,E1 12486.477,E2 12486.477} C_VEL
LIN {X 0,Y 360.791,Z 704.51,A -85,B 0,C 180,E1 12490.39,E2 12490.39} C_VEL
LIN {X 0,Y 359.061,Z 724.58,A -85,B 0,C 180,E1 12494.725,E2 12494.725} C_VEL
LIN {X 0,Y 358.468,Z 740.073,A -85,B 0,C 180,E1 12499.665,E2 12499.665} C_VEL
LIN {X 0,Y 358.668,Z 748.396,A -85,B 0,C 180,E1 12503.964,E2 12503.964} C_VEL
LIN {X 0,Y 358.774,Z 752.009,A -85,B 0,C 180,E1 12507.587,E2 12507.587} C_VEL
LIN {X 0,Y 358.95,Z 752.786,A -85,B 0,C 180,E1 12510.006,E2 12510.006} C_VEL
LIN {X 0,Y 358.649,Z 750.358,A -85,B 0,C 180,E1 12514.849,E2 12514.849} C_VEL
LIN {X 0,Y 358.312,Z 742.625,A -85,B 0,C 180,E1 12519.737,E2 12519.737} C_VEL
LIN {X 0,Y 358.898,Z 728.315,A -85,B 0,C 180,E1 12524.981,E2 12524.981} C_VEL
LIN {X 0,Y 359,Z 727.21,A -85,B 0,C 180,E1 12525.292,E2 12525.292} C_VEL
LIN {X 0,Y 357.208,Z 720.715,A -85,B 0,C 180,E1 12527.093,E2 12527.093} C_VEL
LIN {X 0,Y 353.119,Z 710.166,A -85,B 0,C 180,E1 12529.726,E2 12529.726} C_VEL
LIN {X 0,Y 353.19,Z 708.846,A -85,B 0,C 180,E1 12530.014,E2 12530.014} C_VEL
LIN {X 0,Y 357.202,Z 683.639,A -85,B 0,C 180,E1 12534.549,E2 12534.549} C_VEL
LIN {X 0,Y 362.294,Z 654.467,A -85,B 0,C 180,E1 12538.222,E2 12538.222} C_VEL
LIN {X 0,Y 367.706,Z 621.901,A -85,B 0,C 180,E1 12540.984,E2 12540.984} C_VEL
LIN {X 0,Y 372.018,Z 588.43,A -85,B 0,C 180,E1 12542.758,E2 12542.758} C_VEL
LIN {X 0,Y 371.769,Z 578.832,A -85,B 0,C 180,E1 12543.255,E2 12543.255} C_VEL
LIN {X 0,Y 364.175,Z 557.522,A -85,B 0,C 180,E1 12545.23,E2 12545.23} C_VEL
LIN {X 0,Y 354.321,Z 539.04,A -85,B 0,C 180,E1 12547.967,E2 12547.967} C_VEL
LIN {X 0,Y 349.733,Z 532.276,A -85,B 0,C 180,E1 12549.469,E2 12549.469} C_VEL
LIN {X 0,Y 347.438,Z 526.81,A -85,B 0,C 180,E1 12550.522,E2 12550.522} C_VEL
LIN {X 0,Y 347.395,Z 526.81,A -85,B 0,C 180,E1 12557.818,E2 12557.818} C_VEL
LIN {X 0,Y 347.604,Z 526.81,A -85,B 0,C 180,E1 12565.862,E2 12565.862} C_VEL
LIN {X 0,Y 347.694,Z 527.568,A -85,B 0,C 180,E1 12570.281,E2 12570.281} C_VEL
LIN {X 0,Y 350.766,Z 533.016,A -85,B 0,C 180,E1 12571.583,E2 12571.583} C_VEL
LIN {X 0,Y 359.083,Z 548.847,A -85,B 0,C 180,E1 12574.534,E2 12574.534} C_VEL
LIN {X 0,Y 365.296,Z 568.24,A -85,B 0,C 180,E1 12577.224,E2 12577.224} C_VEL
LIN {X 0,Y 366.517,Z 582.496,A -85,B 0,C 180,E1 12578.89,E2 12578.89} C_VEL
LIN {X 0,Y 362.376,Z 608.083,A -85,B 0,C 180,E1 12581.904,E2 12581.904} C_VEL
LIN {X 0,Y 358.653,Z 627.358,A -85,B 0,C 180,E1 12585.336,E2 12585.336} C_VEL
LIN {X 0,Y 355.558,Z 641.669,A -85,B 0,C 180,E1 12589.326,E2 12589.326} C_VEL
LIN {X 0,Y 353.76,Z 648.649,A -85,B 0,C 180,E1 12592.631,E2 12592.631} C_VEL
LIN {X 0,Y 352.959,Z 651.488,A -85,B 0,C 180,E1 12595.086,E2 12595.086} C_VEL
LIN {X 0,Y 352.289,Z 652.402,A -85,B 0,C 180,E1 12597.545,E2 12597.545} C_VEL
LIN {X 0,Y 351.601,Z 650.312,A -85,B 0,C 180,E1 12601.241,E2 12601.241} C_VEL
LIN {X 0,Y 351.762,Z 642.386,A -85,B 0,C 180,E1 12605.565,E2 12605.565} C_VEL
LIN {X 0,Y 352.451,Z 629.495,A -85,B 0,C 180,E1 12609.453,E2 12609.453} C_VEL
LIN {X 0,Y 353.749,Z 611.654,A -85,B 0,C 180,E1 12612.992,E2 12612.992} C_VEL
LIN {X 0,Y 355.551,Z 587.797,A -85,B 0,C 180,E1 12616.16,E2 12616.16} C_VEL
LIN {X 0,Y 356.255,Z 565.661,A -85,B 0,C 180,E1 12618.192,E2 12618.192} C_VEL
LIN {X 0,Y 350.175,Z 535.559,A -85,B 0,C 180,E1 12620.244,E2 12620.244} C_VEL
LIN {X 0,Y 348.242,Z 526.81,A -85,B 0,C 180,E1 12620.72,E2 12620.72} C_VEL
LIN {X 0,Y 347.712,Z 526.81,A -85,B 0,C 180,E1 12628.626,E2 12628.626} C_VEL
LIN {X 0,Y 347.508,Z 526.81,A -85,B 0,C 180,E1 12634.507,E2 12634.507} C_VEL
LIN {X 0,Y 347.351,Z 526.81,A -85,B 0,C 180,E1 12642.173,E2 12642.173} C_VEL
LIN {X 0,Y 347.405,Z 526.81,A -85,B 0,C 180,E1 12649.169,E2 12649.169} C_VEL
LIN {X 0,Y 347.588,Z 526.81,A -85,B 0,C 180,E1 12655.865,E2 12655.865} C_VEL
LIN {X 0,Y 347.753,Z 526.81,A -85,B 0,C 180,E1 12661.378,E2 12661.378} C_VEL
LIN {X 0,Y 348.121,Z 526.81,A -85,B 0,C 180,E1 12669.632,E2 12669.632} C_VEL
LIN {X 0,Y 348.249,Z 526.81,A -85,B 0,C 180,E1 12674.873,E2 12674.873} C_VEL
LIN {X 0,Y 348.745,Z 526.81,A -85,B 0,C 180,E1 12682.51,E2 12682.51} C_VEL
LIN {X 0,Y 349.258,Z 526.81,A -85,B 0,C 180,E1 12689.994,E2 12689.994} C_VEL
LIN {X 0,Y 348.754,Z 526.81,A -85,B 0,C 180,E1 12697.478,E2 12697.478} C_VEL
LIN {X 0,Y 348.337,Z 526.81,A -85,B 0,C 180,E1 12705.111,E2 12705.111} C_VEL
LIN {X 0,Y 348.133,Z 526.81,A -85,B 0,C 180,E1 12710.354,E2 12710.354} C_VEL
LIN {X 0,Y 347.697,Z 526.81,A -85,B 0,C 180,E1 12718.613,E2 12718.613} C_VEL
LIN {X 0,Y 347.51,Z 526.81,A -85,B 0,C 180,E1 12724.492,E2 12724.492} C_VEL
LIN {X 0,Y 347.32,Z 526.81,A -85,B 0,C 180,E1 12732.168,E2 12732.168} C_VEL
LIN {X 0,Y 347.39,Z 526.81,A -85,B 0,C 180,E1 12739.167,E2 12739.167} C_VEL
LIN {X 0,Y 347.553,Z 526.81,A -85,B 0,C 180,E1 12745.854,E2 12745.854} C_VEL
LIN {X 0,Y 347.727,Z 526.81,A -85,B 0,C 180,E1 12751.375,E2 12751.375} C_VEL
LIN {X 0,Y 348.127,Z 526.81,A -85,B 0,C 180,E1 12759.632,E2 12759.632} C_VEL
LIN {X 0,Y 348.283,Z 526.81,A -85,B 0,C 180,E1 12764.873,E2 12764.873} C_VEL
LIN {X 0,Y 348.775,Z 526.81,A -85,B 0,C 180,E1 12772.51,E2 12772.51} C_VEL
LIN {X 0,Y 349.227,Z 526.81,A -85,B 0,C 180,E1 12779.992,E2 12779.992} C_VEL
LIN {X 0,Y 348.733,Z 526.81,A -85,B 0,C 180,E1 12787.476,E2 12787.476} C_VEL
LIN {X 0,Y 348.286,Z 526.81,A -85,B 0,C 180,E1 12795.111,E2 12795.111} C_VEL
LIN {X 0,Y 348.089,Z 526.81,A -85,B 0,C 180,E1 12800.354,E2 12800.354} C_VEL
LIN {X 0,Y 347.725,Z 526.81,A -85,B 0,C 180,E1 12808.607,E2 12808.607} C_VEL
LIN {X 0,Y 347.576,Z 526.81,A -85,B 0,C 180,E1 12814.481,E2 12814.481} C_VEL
LIN {X 0,Y 347.283,Z 526.81,A -85,B 0,C 180,E1 12822.179,E2 12822.179} C_VEL
LIN {X 0,Y 347.253,Z 526.81,A -85,B 0,C 180,E1 12829.162,E2 12829.162} C_VEL
LIN {X 0,Y 347.685,Z 526.81,A -85,B 0,C 180,E1 12837.003,E2 12837.003} C_VEL
LIN {X 0,Y 364.94,Z 583.605,A -85,B 0,C 180,E1 12839.389,E2 12839.389} C_VEL
LIN {X 0,Y 362.626,Z 616.928,A -85,B 0,C 180,E1 12840.779,E2 12840.779} C_VEL
LIN {X 0,Y 359.397,Z 648.972,A -85,B 0,C 180,E1 12843.078,E2 12843.078} C_VEL
LIN {X 0,Y 356.063,Z 677.93,A -85,B 0,C 180,E1 12846.211,E2 12846.211} C_VEL
LIN {X 0,Y 352.999,Z 703.618,A -85,B 0,C 180,E1 12850.202,E2 12850.202} C_VEL
LIN {X 0,Y 351.193,Z 723.895,A -85,B 0,C 180,E1 12854.695,E2 12854.695} C_VEL
LIN {X 0,Y 350.673,Z 738.491,A -85,B 0,C 180,E1 12859.432,E2 12859.432} C_VEL
LIN {X 0,Y 350.878,Z 747.291,A -85,B 0,C 180,E1 12864.032,E2 12864.032} C_VEL
LIN {X 0,Y 350.983,Z 750.724,A -85,B 0,C 180,E1 12867.533,E2 12867.533} C_VEL
LIN {X 0,Y 351.163,Z 751.57,A -85,B 0,C 180,E1 12870.006,E2 12870.006} C_VEL
LIN {X 0,Y 350.813,Z 749.205,A -85,B 0,C 180,E1 12874.958,E2 12874.958} C_VEL
LIN {X 0,Y 350.428,Z 741.562,A -85,B 0,C 180,E1 12879.958,E2 12879.958} C_VEL
LIN {X 0,Y 351.14,Z 727.156,A -85,B 0,C 180,E1 12885.377,E2 12885.377} C_VEL
LIN {X 0,Y 353.19,Z 708.846,A -85,B 0,C 180,E1 12890.014,E2 12890.014} C_VEL
LIN {X 0,Y 351.072,Z 698.411,A -85,B 0,C 180,E1 12892.279,E2 12892.279} C_VEL
LIN {X 0,Y 349.253,Z 687.178,A -85,B 0,C 180,E1 12894.464,E2 12894.464} C_VEL
LIN {X 0,Y 354.588,Z 658.269,A -85,B 0,C 180,E1 12898.431,E2 12898.431} C_VEL
LIN {X 0,Y 360.437,Z 626.981,A -85,B 0,C 180,E1 12901.328,E2 12901.328} C_VEL
LIN {X 0,Y 365.374,Z 593.236,A -85,B 0,C 180,E1 12903.339,E2 12903.339} C_VEL
LIN {X 0,Y 365.94,Z 582.344,A -85,B 0,C 180,E1 12903.871,E2 12903.871} C_VEL
LIN {X 0,Y 359.127,Z 562.102,A -85,B 0,C 180,E1 12905.876,E2 12905.876} C_VEL
LIN {X 0,Y 350.321,Z 545.056,A -85,B 0,C 180,E1 12908.522,E2 12908.522} C_VEL
LIN {X 0,Y 342.8,Z 533.213,A -85,B 0,C 180,E1 12911.436,E2 12911.436} C_VEL
LIN {X 0,Y 339.54,Z 527.83,A -85,B 0,C 180,E1 12913.206,E2 12913.206} C_VEL
LIN {X 0,Y 339.485,Z 526.81,A -85,B 0,C 180,E1 12913.664,E2 12913.664} C_VEL
LIN {X 0,Y 339.479,Z 526.81,A -85,B 0,C 180,E1 12921.375,E2 12921.375} C_VEL
LIN {X 0,Y 339.688,Z 527.532,A -85,B 0,C 180,E1 12927.515,E2 12927.515} C_VEL
LIN {X 0,Y 343.167,Z 533.272,A -85,B 0,C 180,E1 12929.475,E2 12929.475} C_VEL
LIN {X 0,Y 350.767,Z 546.917,A -85,B 0,C 180,E1 12932.718,E2 12932.718} C_VEL
LIN {X 0,Y 358.193,Z 566.695,A -85,B 0,C 180,E1 12935.966,E2 12935.966} C_VEL
LIN {X 0,Y 360.308,Z 583.419,A -85,B 0,C 180,E1 12938.122,E2 12938.122} C_VEL
LIN {X 0,Y 355.914,Z 608.257,A -85,B 0,C 180,E1 12941.082,E2 12941.082} C_VEL
LIN {X 0,Y 352.015,Z 627.123,A -85,B 0,C 180,E1 12944.415,E2 12944.415} C_VEL
LIN {X 0,Y 348.616,Z 641.263,A -85,B 0,C 180,E1 12948.215,E2 12948.215} C_VEL
LIN {X 0,Y 346.117,Z 650.384,A -85,B 0,C 180,E1 12952.467,E2 12952.467} C_VEL
LIN {X 0,Y 345.229,Z 652.972,A -85,B 0,C 180,E1 12954.976,E2 12954.976} C_VEL
LIN {X 0,Y 344.511,Z 653.737,A -85,B 0,C 180,E1 12957.489,E2 12957.489} C_VEL
LIN {X 0,Y 343.783,Z 651.358,A -85,B 0,C 180,E1 12961.27,E2 12961.27} C_VEL
LIN {X 0,Y 343.945,Z 643.117,A -85,B 0,C 180,E1 12965.692,E2 12965.692} C_VEL
LIN {X 0,Y 344.678,Z 629.398,A -85,B 0,C 180,E1 12969.786,E2 12969.786} C_VEL
LIN {X 0,Y 346.171,Z 609.572,A -85,B 0,C 180,E1 12973.604,E2 12973.604} C_VEL
LIN {X 0,Y 348.062,Z 585.04,A -85,B 0,C 180,E1 12976.75,E2 12976.75} C_VEL
LIN {X 0,Y 348.518,Z 566.742,A -85,B 0,C 180,E1 12978.431,E2 12978.431} C_VEL
LIN {X 0,Y 342.409,Z 536.405,A -85,B 0,C 180,E1 12980.548,E2 12980.548} C_VEL
LIN {X 0,Y 340.273,Z 526.81,A -85,B 0,C 180,E1 12981.167,E2 12981.167} C_VEL
LIN {X 0,Y 339.763,Z 526.81,A -85,B 0,C 180,E1 12989.36,E2 12989.36} C_VEL
LIN {X 0,Y 339.43,Z 526.81,A -85,B 0,C 180,E1 12996.581,E2 12996.581} C_VEL
LIN {X 0,Y 339.477,Z 526.81,A -85,B 0,C 180,E1 13004.463,E2 13004.463} C_VEL
LIN {X 0,Y 339.487,Z 526.81,A -85,B 0,C 180,E1 13011.356,E2 13011.356} C_VEL
LIN {X 0,Y 339.696,Z 526.81,A -85,B 0,C 180,E1 13017.881,E2 13017.881} C_VEL
LIN {X 0,Y 339.863,Z 526.81,A -85,B 0,C 180,E1 13023.538,E2 13023.538} C_VEL
LIN {X 0,Y 340.157,Z 526.81,A -85,B 0,C 180,E1 13029.198,E2 13029.198} C_VEL
LIN {X 0,Y 340.427,Z 526.81,A -85,B 0,C 180,E1 13037.145,E2 13037.145} C_VEL
LIN {X 0,Y 340.977,Z 526.81,A -85,B 0,C 180,E1 13044.899,E2 13044.899} C_VEL
LIN {X 0,Y 341.371,Z 526.81,A -85,B 0,C 180,E1 13049.994,E2 13049.994} C_VEL
LIN {X 0,Y 340.819,Z 526.81,A -85,B 0,C 180,E1 13057.653,E2 13057.653} C_VEL
LIN {X 0,Y 340.41,Z 526.81,A -85,B 0,C 180,E1 13065.472,E2 13065.472} C_VEL
LIN {X 0,Y 340.165,Z 526.81,A -85,B 0,C 180,E1 13070.853,E2 13070.853} C_VEL
LIN {X 0,Y 339.751,Z 526.81,A -85,B 0,C 180,E1 13079.347,E2 13079.347} C_VEL
LIN {X 0,Y 339.417,Z 526.81,A -85,B 0,C 180,E1 13086.579,E2 13086.579} C_VEL
LIN {X 0,Y 339.447,Z 526.81,A -85,B 0,C 180,E1 13094.458,E2 13094.458} C_VEL
LIN {X 0,Y 339.468,Z 526.81,A -85,B 0,C 180,E1 13101.353,E2 13101.353} C_VEL
LIN {X 0,Y 339.676,Z 526.81,A -85,B 0,C 180,E1 13107.865,E2 13107.865} C_VEL
LIN {X 0,Y 339.84,Z 526.81,A -85,B 0,C 180,E1 13113.536,E2 13113.536} C_VEL
LIN {X 0,Y 340.299,Z 526.81,A -85,B 0,C 180,E1 13121.846,E2 13121.846} C_VEL
LIN {X 0,Y 340.586,Z 526.81,A -85,B 0,C 180,E1 13129.75,E2 13129.75} C_VEL
LIN {X 0,Y 341.237,Z 526.81,A -85,B 0,C 180,E1 13137.449,E2 13137.449} C_VEL
LIN {X 0,Y 341.223,Z 526.81,A -85,B 0,C 180,E1 13142.535,E2 13142.535} C_VEL
LIN {X 0,Y 340.599,Z 526.81,A -85,B 0,C 180,E1 13150.234,E2 13150.234} C_VEL
LIN {X 0,Y 340.268,Z 526.81,A -85,B 0,C 180,E1 13158.139,E2 13158.139} C_VEL
LIN {X 0,Y 339.823,Z 526.81,A -85,B 0,C 180,E1 13166.448,E2 13166.448} C_VEL
LIN {X 0,Y 339.711,Z 526.81,A -85,B 0,C 180,E1 13172.321,E2 13172.321} C_VEL
LIN {X 0,Y 339.439,Z 526.81,A -85,B 0,C 180,E1 13178.631,E2 13178.631} C_VEL
LIN {X 0,Y 339.356,Z 526.81,A -85,B 0,C 180,E1 13185.535,E2 13185.535} C_VEL
LIN {X 0,Y 339.374,Z 526.81,A -85,B 0,C 180,E1 13193.405,E2 13193.405} C_VEL
LIN {X 0,Y 339.729,Z 526.976,A -85,B 0,C 180,E1 13196.561,E2 13196.561} C_VEL
LIN {X 0,Y 357.312,Z 585.871,A -85,B 0,C 180,E1 13199.091,E2 13199.091} C_VEL
LIN {X 0,Y 354.698,Z 620.068,A -85,B 0,C 180,E1 13200.641,E2 13200.641} C_VEL
LIN {X 0,Y 351.315,Z 651.94,A -85,B 0,C 180,E1 13203.101,E2 13203.101} C_VEL
LIN {X 0,Y 347.932,Z 680.422,A -85,B 0,C 180,E1 13206.39,E2 13206.39} C_VEL
LIN {X 0,Y 344.894,Z 705.379,A -85,B 0,C 180,E1 13210.523,E2 13210.523} C_VEL
LIN {X 0,Y 343.246,Z 724.663,A -85,B 0,C 180,E1 13215.084,E2 13215.084} C_VEL
LIN {X 0,Y 342.835,Z 738.386,A -85,B 0,C 180,E1 13219.831,E2 13219.831} C_VEL
LIN {X 0,Y 343.071,Z 746.17,A -85,B 0,C 180,E1 13224.119,E2 13224.119} C_VEL
LIN {X 0,Y 343.172,Z 749.418,A -85,B 0,C 180,E1 13227.477,E2 13227.477} C_VEL
LIN {X 0,Y 343.352,Z 750.341,A -85,B 0,C 180,E1 13230.006,E2 13230.006} C_VEL
LIN {X 0,Y 342.983,Z 748.054,A -85,B 0,C 180,E1 13235.071,E2 13235.071} C_VEL
LIN {X 0,Y 342.562,Z 740.519,A -85,B 0,C 180,E1 13240.189,E2 13240.189} C_VEL
LIN {X 0,Y 343.354,Z 726.399,A -85,B 0,C 180,E1 13245.676,E2 13245.676} C_VEL
LIN {X 0,Y 345.816,Z 706.428,A -85,B 0,C 180,E1 13250.845,E2 13250.845} C_VEL
LIN {X 0,Y 349.253,Z 687.178,A -85,B 0,C 180,E1 13254.464,E2 13254.464} C_VEL
LIN {X 0,Y 347.911,Z 675.337,A -85,B 0,C 180,E1 13256.584,E2 13256.584} C_VEL
LIN {X 0,Y 346.846,Z 662.567,A -85,B 0,C 180,E1 13258.55,E2 13258.55} C_VEL
LIN {X 0,Y 353.061,Z 631.728,A -85,B 0,C 180,E1 13261.697,E2 13261.697} C_VEL
LIN {X 0,Y 358.674,Z 598.105,A -85,B 0,C 180,E1 13263.922,E2 13263.922} C_VEL
LIN {X 0,Y 359.913,Z 584.409,A -85,B 0,C 180,E1 13264.635,E2 13264.635} C_VEL
LIN {X 0,Y 353.138,Z 564.323,A -85,B 0,C 180,E1 13266.867,E2 13266.867} C_VEL
LIN {X 0,Y 345.232,Z 549.154,A -85,B 0,C 180,E1 13269.514,E2 13269.514} C_VEL
LIN {X 0,Y 339.571,Z 540.061,A -85,B 0,C 180,E1 13271.943,E2 13271.943} C_VEL
LIN {X 0,Y 335.594,Z 533.677,A -85,B 0,C 180,E1 13274.342,E2 13274.342} C_VEL
LIN {X 0,Y 331.597,Z 527.659,A -85,B 0,C 180,E1 13279.747,E2 13279.747} C_VEL
LIN {X 0,Y 332.098,Z 529.635,A -85,B 0,C 180,E1 13283.064,E2 13283.064} C_VEL
LIN {X 0,Y 336.615,Z 535.094,A -85,B 0,C 180,E1 13287.201,E2 13287.201} C_VEL
LIN {X 0,Y 341.239,Z 543.388,A -85,B 0,C 180,E1 13289.908,E2 13289.908} C_VEL
LIN {X 0,Y 347.458,Z 555.289,A -85,B 0,C 180,E1 13292.74,E2 13292.74} C_VEL
LIN {X 0,Y 352.935,Z 573.009,A -85,B 0,C 180,E1 13295.711,E2 13295.711} C_VEL
LIN {X 0,Y 353.918,Z 586.703,A -85,B 0,C 180,E1 13297.535,E2 13297.535} C_VEL
LIN {X 0,Y 348.994,Z 611.743,A -85,B 0,C 180,E1 13300.692,E2 13300.692} C_VEL
LIN {X 0,Y 344.475,Z 631.134,A -85,B 0,C 180,E1 13304.392,E2 13304.392} C_VEL
LIN {X 0,Y 340.851,Z 644.754,A -85,B 0,C 180,E1 13308.468,E2 13308.468} C_VEL
LIN {X 0,Y 338.493,Z 652.098,A -85,B 0,C 180,E1 13312.297,E2 13312.297} C_VEL
LIN {X 0,Y 337.521,Z 654.482,A -85,B 0,C 180,E1 13314.861,E2 13314.861} C_VEL
LIN {X 0,Y 336.76,Z 655.069,A -85,B 0,C 180,E1 13317.431,E2 13317.431} C_VEL
LIN {X 0,Y 335.984,Z 652.396,A -85,B 0,C 180,E1 13321.299,E2 13321.299} C_VEL
LIN {X 0,Y 336.103,Z 643.771,A -85,B 0,C 180,E1 13325.825,E2 13325.825} C_VEL
LIN {X 0,Y 336.894,Z 629.806,A -85,B 0,C 180,E1 13330.004,E2 13330.004} C_VEL
LIN {X 0,Y 338.464,Z 609.454,A -85,B 0,C 180,E1 13333.92,E2 13333.92} C_VEL
LIN {X 0,Y 340.417,Z 584.285,A -85,B 0,C 180,E1 13337.138,E2 13337.138} C_VEL
LIN {X 0,Y 340.83,Z 567.943,A -85,B 0,C 180,E1 13338.65,E2 13338.65} C_VEL
LIN {X 0,Y 334.678,Z 537.427,A -85,B 0,C 180,E1 13340.858,E2 13340.858} C_VEL
LIN {X 0,Y 332.297,Z 526.81,A -85,B 0,C 180,E1 13341.488,E2 13341.488} C_VEL
LIN {X 0,Y 331.78,Z 526.81,A -85,B 0,C 180,E1 13349.869,E2 13349.869} C_VEL
LIN {X 0,Y 331.555,Z 526.81,A -85,B 0,C 180,E1 13356.425,E2 13356.425} C_VEL
LIN {X 0,Y 331.502,Z 526.81,A -85,B 0,C 180,E1 13363.251,E2 13363.251} C_VEL
LIN {X 0,Y 331.576,Z 526.81,A -85,B 0,C 180,E1 13370.929,E2 13370.929} C_VEL
LIN {X 0,Y 331.632,Z 526.81,A -85,B 0,C 180,E1 13376.772,E2 13376.772} C_VEL
LIN {X 0,Y 331.925,Z 526.81,A -85,B 0,C 180,E1 13382.854,E2 13382.854} C_VEL
LIN {X 0,Y 332.292,Z 526.81,A -85,B 0,C 180,E1 13391.394,E2 13391.394} C_VEL
LIN {X 0,Y 332.653,Z 526.81,A -85,B 0,C 180,E1 13399.504,E2 13399.504} C_VEL
LIN {X 0,Y 333.376,Z 526.81,A -85,B 0,C 180,E1 13407.391,E2 13407.391} C_VEL
LIN {X 0,Y 333.308,Z 526.81,A -85,B 0,C 180,E1 13412.597,E2 13412.597} C_VEL
LIN {X 0,Y 332.727,Z 526.81,A -85,B 0,C 180,E1 13420.481,E2 13420.481} C_VEL
LIN {X 0,Y 332.334,Z 526.81,A -85,B 0,C 180,E1 13428.591,E2 13428.591} C_VEL
LIN {X 0,Y 331.88,Z 526.81,A -85,B 0,C 180,E1 13437.136,E2 13437.136} C_VEL
LIN {X 0,Y 331.537,Z 526.81,A -85,B 0,C 180,E1 13444.702,E2 13444.702} C_VEL
LIN {X 0,Y 331.493,Z 526.81,A -85,B 0,C 180,E1 13449.742,E2 13449.742} C_VEL
LIN {X 0,Y 331.502,Z 526.81,A -85,B 0,C 180,E1 13456.942,E2 13456.942} C_VEL
LIN {X 0,Y 331.578,Z 526.81,A -85,B 0,C 180,E1 13463.578,E2 13463.578} C_VEL
LIN {X 0,Y 331.831,Z 526.81,A -85,B 0,C 180,E1 13470.091,E2 13470.091} C_VEL
LIN {X 0,Y 332.143,Z 526.81,A -85,B 0,C 180,E1 13478.605,E2 13478.605} C_VEL
LIN {X 0,Y 332.409,Z 526.81,A -85,B 0,C 180,E1 13484.132,E2 13484.132} C_VEL
LIN {X 0,Y 332.899,Z 526.81,A -85,B 0,C 180,E1 13492.15,E2 13492.15} C_VEL
LIN {X 0,Y 333.436,Z 526.81,A -85,B 0,C 180,E1 13499.992,E2 13499.992} C_VEL
LIN {X 0,Y 332.867,Z 526.81,A -85,B 0,C 180,E1 13507.834,E2 13507.834} C_VEL
LIN {X 0,Y 332.401,Z 526.81,A -85,B 0,C 180,E1 13515.851,E2 13515.851} C_VEL
LIN {X 0,Y 332.111,Z 526.81,A -85,B 0,C 180,E1 13521.38,E2 13521.38} C_VEL
LIN {X 0,Y 331.812,Z 526.81,A -85,B 0,C 180,E1 13529.903,E2 13529.903} C_VEL
LIN {X 0,Y 331.576,Z 526.81,A -85,B 0,C 180,E1 13536.402,E2 13536.402} C_VEL
LIN {X 0,Y 331.403,Z 526.81,A -85,B 0,C 180,E1 13543.245,E2 13543.245} C_VEL
LIN {X 0,Y 331.438,Z 526.81,A -85,B 0,C 180,E1 13550.933,E2 13550.933} C_VEL
LIN {X 0,Y 331.811,Z 526.967,A -85,B 0,C 180,E1 13556.088,E2 13556.088} C_VEL
LIN {X 0,Y 349.749,Z 585.733,A -85,B 0,C 180,E1 13558.709,E2 13558.709} C_VEL
LIN {X 0,Y 347.175,Z 618.985,A -85,B 0,C 180,E1 13560.252,E2 13560.252} C_VEL
LIN {X 0,Y 343.624,Z 651.365,A -85,B 0,C 180,E1 13562.804,E2 13562.804} C_VEL
LIN {X 0,Y 340.188,Z 679.637,A -85,B 0,C 180,E1 13566.145,E2 13566.145} C_VEL
LIN {X 0,Y 337.09,Z 704.567,A -85,B 0,C 180,E1 13570.37,E2 13570.37} C_VEL
LIN {X 0,Y 335.392,Z 723.713,A -85,B 0,C 180,E1 13575.019,E2 13575.019} C_VEL
LIN {X 0,Y 335.016,Z 738.179,A -85,B 0,C 180,E1 13580.249,E2 13580.249} C_VEL
LIN {X 0,Y 335.285,Z 745.76,A -85,B 0,C 180,E1 13584.824,E2 13584.824} C_VEL
LIN {X 0,Y 335.564,Z 749.107,A -85,B 0,C 180,E1 13590.006,E2 13590.006} C_VEL
LIN {X 0,Y 335.138,Z 746.903,A -85,B 0,C 180,E1 13595.19,E2 13595.19} C_VEL
LIN {X 0,Y 334.701,Z 739.469,A -85,B 0,C 180,E1 13600.431,E2 13600.431} C_VEL
LIN {X 0,Y 335.452,Z 726.478,A -85,B 0,C 180,E1 13605.719,E2 13605.719} C_VEL
LIN {X 0,Y 338.003,Z 707.21,A -85,B 0,C 180,E1 13611.006,E2 13611.006} C_VEL
LIN {X 0,Y 342.655,Z 682.929,A -85,B 0,C 180,E1 13615.664,E2 13615.664} C_VEL
LIN {X 0,Y 346.846,Z 662.567,A -85,B 0,C 180,E1 13618.55,E2 13618.55} C_VEL
LIN {X 0,Y 345.702,Z 637.101,A -85,B 0,C 180,E1 13621.985,E2 13621.985} C_VEL
LIN {X 0,Y 346.019,Z 635.21,A -85,B 0,C 180,E1 13622.165,E2 13622.165} C_VEL
LIN {X 0,Y 352.215,Z 602.14,A -85,B 0,C 180,E1 13624.561,E2 13624.561} C_VEL
LIN {X 0,Y 353.899,Z 586.564,A -85,B 0,C 180,E1 13625.443,E2 13625.443} C_VEL
LIN {X 0,Y 347.802,Z 567.761,A -85,B 0,C 180,E1 13627.762,E2 13627.762} C_VEL
LIN {X 0,Y 340.21,Z 552.732,A -85,B 0,C 180,E1 13630.659,E2 13630.659} C_VEL
LIN {X 0,Y 335.529,Z 545.66,A -85,B 0,C 180,E1 13632.928,E2 13632.928} C_VEL
LIN {X 0,Y 332.956,Z 540.945,A -85,B 0,C 180,E1 13634.725,E2 13634.725} C_VEL
LIN {X 0,Y 329.456,Z 535.216,A -85,B 0,C 180,E1 13639.968,E2 13639.968} C_VEL
LIN {X 0,Y 330.27,Z 538.22,A -85,B 0,C 180,E1 13643.815,E2 13643.815} C_VEL
LIN {X 0,Y 333.714,Z 542.52,A -85,B 0,C 180,E1 13646.928,E2 13646.928} C_VEL
LIN {X 0,Y 339.171,Z 552.381,A -85,B 0,C 180,E1 13650.242,E2 13650.242} C_VEL
LIN {X 0,Y 345.467,Z 569.178,A -85,B 0,C 180,E1 13653.809,E2 13653.809} C_VEL
LIN {X 0,Y 348.024,Z 586.476,A -85,B 0,C 180,E1 13656.504,E2 13656.504} C_VEL
LIN {X 0,Y 342.984,Z 611.314,A -85,B 0,C 180,E1 13659.667,E2 13659.667} C_VEL
LIN {X 0,Y 338.005,Z 631.186,A -85,B 0,C 180,E1 13663.417,E2 13663.417} C_VEL
LIN {X 0,Y 333.731,Z 645.816,A -85,B 0,C 180,E1 13667.772,E2 13667.772} C_VEL
LIN {X 0,Y 330.881,Z 653.827,A -85,B 0,C 180,E1 13672.118,E2 13672.118} C_VEL
LIN {X 0,Y 329.81,Z 655.997,A -85,B 0,C 180,E1 13674.74,E2 13674.74} C_VEL
LIN {X 0,Y 328.981,Z 656.369,A -85,B 0,C 180,E1 13677.37,E2 13677.37} C_VEL
LIN {X 0,Y 328.162,Z 653.428,A -85,B 0,C 180,E1 13681.33,E2 13681.33} C_VEL
LIN {X 0,Y 328.267,Z 644.605,A -85,B 0,C 180,E1 13685.891,E2 13685.891} C_VEL
LIN {X 0,Y 329.104,Z 629.873,A -85,B 0,C 180,E1 13690.277,E2 13690.277} C_VEL
LIN {X 0,Y 330.78,Z 609.236,A -85,B 0,C 180,E1 13694.25,E2 13694.25} C_VEL
LIN {X 0,Y 332.78,Z 584.104,A -85,B 0,C 180,E1 13697.474,E2 13697.474} C_VEL
LIN {X 0,Y 332.929,Z 568.17,A -85,B 0,C 180,E1 13698.975,E2 13698.975} C_VEL
LIN {X 0,Y 326.916,Z 538.214,A -85,B 0,C 180,E1 13701.185,E2 13701.185} C_VEL
LIN {X 0,Y 324.343,Z 526.81,A -85,B 0,C 180,E1 13701.936,E2 13701.936} C_VEL
LIN {X 0,Y 323.91,Z 526.81,A -85,B 0,C 180,E1 13707.876,E2 13707.876} C_VEL
LIN {X 0,Y 323.629,Z 526.81,A -85,B 0,C 180,E1 13714.161,E2 13714.161} C_VEL
LIN {X 0,Y 323.476,Z 526.81,A -85,B 0,C 180,E1 13721.495,E2 13721.495} C_VEL
LIN {X 0,Y 323.517,Z 526.81,A -85,B 0,C 180,E1 13729.057,E2 13729.057} C_VEL
LIN {X 0,Y 323.678,Z 526.81,A -85,B 0,C 180,E1 13735.845,E2 13735.845} C_VEL
LIN {X 0,Y 323.987,Z 526.81,A -85,B 0,C 180,E1 13742.625,E2 13742.625} C_VEL
LIN {X 0,Y 324.309,Z 526.81,A -85,B 0,C 180,E1 13750.919,E2 13750.919} C_VEL
LIN {X 0,Y 324.702,Z 526.81,A -85,B 0,C 180,E1 13759.244,E2 13759.244} C_VEL
LIN {X 0,Y 325.454,Z 526.81,A -85,B 0,C 180,E1 13767.327,E2 13767.327} C_VEL
LIN {X 0,Y 325.392,Z 526.81,A -85,B 0,C 180,E1 13772.661,E2 13772.661} C_VEL
LIN {X 0,Y 324.78,Z 526.81,A -85,B 0,C 180,E1 13780.741,E2 13780.741} C_VEL
LIN {X 0,Y 324.347,Z 526.81,A -85,B 0,C 180,E1 13789.066,E2 13789.066} C_VEL
LIN {X 0,Y 323.954,Z 526.81,A -85,B 0,C 180,E1 13797.364,E2 13797.364} C_VEL
LIN {X 0,Y 323.631,Z 526.81,A -85,B 0,C 180,E1 13804.145,E2 13804.145} C_VEL
LIN {X 0,Y 323.442,Z 526.81,A -85,B 0,C 180,E1 13811.489,E2 13811.489} C_VEL
LIN {X 0,Y 323.497,Z 526.81,A -85,B 0,C 180,E1 13819.054,E2 13819.054} C_VEL
LIN {X 0,Y 323.656,Z 526.81,A -85,B 0,C 180,E1 13825.842,E2 13825.842} C_VEL
LIN {X 0,Y 323.99,Z 526.81,A -85,B 0,C 180,E1 13832.597,E2 13832.597} C_VEL
LIN {X 0,Y 324.331,Z 526.81,A -85,B 0,C 180,E1 13840.919,E2 13840.919} C_VEL
LIN {X 0,Y 324.7,Z 526.81,A -85,B 0,C 180,E1 13849.242,E2 13849.242} C_VEL
LIN {X 0,Y 325.402,Z 526.81,A -85,B 0,C 180,E1 13857.325,E2 13857.325} C_VEL
LIN {X 0,Y 325.397,Z 526.81,A -85,B 0,C 180,E1 13862.659,E2 13862.659} C_VEL
LIN {X 0,Y 324.722,Z 526.81,A -85,B 0,C 180,E1 13870.74,E2 13870.74} C_VEL
LIN {X 0,Y 324.3,Z 526.81,A -85,B 0,C 180,E1 13879.066,E2 13879.066} C_VEL
LIN {X 0,Y 323.948,Z 526.81,A -85,B 0,C 180,E1 13887.388,E2 13887.388} C_VEL
LIN {X 0,Y 323.688,Z 526.81,A -85,B 0,C 180,E1 13894.134,E2 13894.134} C_VEL
LIN {X 0,Y 323.407,Z 526.81,A -85,B 0,C 180,E1 13901.501,E2 13901.501} C_VEL
LIN {X 0,Y 323.378,Z 526.81,A -85,B 0,C 180,E1 13909.052,E2 13909.052} C_VEL
LIN {X 0,Y 323.867,Z 527.313,A -85,B 0,C 180,E1 13915.624,E2 13915.624} C_VEL
LIN {X 0,Y 342.086,Z 588.508,A -85,B 0,C 180,E1 13918.425,E2 13918.425} C_VEL
LIN {X 0,Y 339.117,Z 622.667,A -85,B 0,C 180,E1 13920.169,E2 13920.169} C_VEL
LIN {X 0,Y 335.574,Z 653.873,A -85,B 0,C 180,E1 13922.824,E2 13922.824} C_VEL
LIN {X 0,Y 331.876,Z 682.67,A -85,B 0,C 180,E1 13926.479,E2 13926.479} C_VEL
LIN {X 0,Y 328.926,Z 707.038,A -85,B 0,C 180,E1 13930.946,E2 13930.946} C_VEL
LIN {X 0,Y 327.444,Z 725.528,A -85,B 0,C 180,E1 13935.821,E2 13935.821} C_VEL
LIN {X 0,Y 327.185,Z 737.927,A -85,B 0,C 180,E1 13940.685,E2 13940.685} C_VEL
LIN {X 0,Y 327.512,Z 745.699,A -85,B 0,C 180,E1 13946.03,E2 13946.03} C_VEL
LIN {X 0,Y 327.759,Z 747.834,A -85,B 0,C 180,E1 13950.006,E2 13950.006} C_VEL
LIN {X 0,Y 327.273,Z 745.752,A -85,B 0,C 180,E1 13955.315,E2 13955.315} C_VEL
LIN {X 0,Y 326.841,Z 738.416,A -85,B 0,C 180,E1 13960.685,E2 13960.685} C_VEL
LIN {X 0,Y 327.677,Z 725.614,A -85,B 0,C 180,E1 13966.102,E2 13966.102} C_VEL
LIN {X 0,Y 330.459,Z 706.628,A -85,B 0,C 180,E1 13971.509,E2 13971.509} C_VEL
LIN {X 0,Y 335.418,Z 683.031,A -85,B 0,C 180,E1 13976.214,E2 13976.214} C_VEL
LIN {X 0,Y 341.854,Z 654.082,A -85,B 0,C 180,E1 13980.255,E2 13980.255} C_VEL
LIN {X 0,Y 346.019,Z 635.21,A -85,B 0,C 180,E1 13982.165,E2 13982.165} C_VEL
LIN {X 0,Y 345.976,Z 620.706,A -85,B 0,C 180,E1 13983.808,E2 13983.808} C_VEL
LIN {X 0,Y 345.571,Z 607.642,A -85,B 0,C 180,E1 13985.133,E2 13985.133} C_VEL
LIN {X 0,Y 345.86,Z 605.633,A -85,B 0,C 180,E1 13985.266,E2 13985.266} C_VEL
LIN {X 0,Y 348.125,Z 588.997,A -85,B 0,C 180,E1 13986.273,E2 13986.273} C_VEL
LIN {X 0,Y 342.454,Z 570.556,A -85,B 0,C 180,E1 13988.79,E2 13988.79} C_VEL
LIN {X 0,Y 335.231,Z 556.541,A -85,B 0,C 180,E1 13991.959,E2 13991.959} C_VEL
LIN {X 0,Y 330.22,Z 548.119,A -85,B 0,C 180,E1 13995.206,E2 13995.206} C_VEL
LIN {X 0,Y 327.37,Z 542.916,A -85,B 0,C 180,E1 13999.66,E2 13999.66} C_VEL
LIN {X 0,Y 327.523,Z 544.773,A -85,B 0,C 180,E1 14002.864,E2 14002.864} C_VEL
LIN {X 0,Y 330.782,Z 549.63,A -85,B 0,C 180,E1 14006.56,E2 14006.56} C_VEL
LIN {X 0,Y 336.045,Z 560.692,A -85,B 0,C 180,E1 14010.301,E2 14010.301} C_VEL
LIN {X 0,Y 341.066,Z 577.876,A -85,B 0,C 180,E1 14013.941,E2 14013.941} C_VEL
LIN {X 0,Y 341.793,Z 591.427,A -85,B 0,C 180,E1 14016.049,E2 14016.049} C_VEL
LIN {X 0,Y 336.191,Z 615.088,A -85,B 0,C 180,E1 14019.237,E2 14019.237} C_VEL
LIN {X 0,Y 330.522,Z 635.321,A -85,B 0,C 180,E1 14023.373,E2 14023.373} C_VEL
LIN {X 0,Y 326.312,Z 648.059,A -85,B 0,C 180,E1 14027.521,E2 14027.521} C_VEL
LIN {X 0,Y 323.247,Z 655.554,A -85,B 0,C 180,E1 14031.931,E2 14031.931} C_VEL
LIN {X 0,Y 322.106,Z 657.544,A -85,B 0,C 180,E1 14034.614,E2 14034.614} C_VEL
LIN {X 0,Y 321.205,Z 657.644,A -85,B 0,C 180,E1 14037.307,E2 14037.307} C_VEL
LIN {X 0,Y 320.266,Z 653.428,A -85,B 0,C 180,E1 14042.04,E2 14042.04} C_VEL
LIN {X 0,Y 320.478,Z 643.453,A -85,B 0,C 180,E1 14046.688,E2 14046.688} C_VEL
LIN {X 0,Y 321.417,Z 628.581,A -85,B 0,C 180,E1 14050.869,E2 14050.869} C_VEL
LIN {X 0,Y 323.135,Z 607.711,A -85,B 0,C 180,E1 14054.768,E2 14054.768} C_VEL
LIN {X 0,Y 325.162,Z 582.389,A -85,B 0,C 180,E1 14057.958,E2 14057.958} C_VEL
LIN {X 0,Y 325.25,Z 569.565,A -85,B 0,C 180,E1 14059.181,E2 14059.181} C_VEL
LIN {X 0,Y 319.153,Z 538.989,A -85,B 0,C 180,E1 14061.505,E2 14061.505} C_VEL
LIN {X 0,Y 316.366,Z 526.81,A -85,B 0,C 180,E1 14062.283,E2 14062.283} C_VEL
LIN {X 0,Y 315.78,Z 526.81,A -85,B 0,C 180,E1 14070.327,E2 14070.327} C_VEL
LIN {X 0,Y 315.519,Z 526.81,A -85,B 0,C 180,E1 14078.605,E2 14078.605} C_VEL
LIN {X 0,Y 315.493,Z 526.81,A -85,B 0,C 180,E1 14086.052,E2 14086.052} C_VEL
LIN {X 0,Y 315.557,Z 526.81,A -85,B 0,C 180,E1 14091.401,E2 14091.401} C_VEL
LIN {X 0,Y 315.83,Z 526.81,A -85,B 0,C 180,E1 14099.656,E2 14099.656} C_VEL
LIN {X 0,Y 316.181,Z 526.81,A -85,B 0,C 180,E1 14107.468,E2 14107.468} C_VEL
LIN {X 0,Y 316.479,Z 526.81,A -85,B 0,C 180,E1 14113.312,E2 14113.312} C_VEL
LIN {X 0,Y 316.99,Z 526.81,A -85,B 0,C 180,E1 14121.755,E2 14121.755} C_VEL
LIN {X 0,Y 317.545,Z 526.81,A -85,B 0,C 180,E1 14127.261,E2 14127.261} C_VEL
LIN {X 0,Y 317.503,Z 526.81,A -85,B 0,C 180,E1 14132.727,E2 14132.727} C_VEL
LIN {X 0,Y 316.859,Z 526.81,A -85,B 0,C 180,E1 14141.012,E2 14141.012} C_VEL
LIN {X 0,Y 316.399,Z 526.81,A -85,B 0,C 180,E1 14149.564,E2 14149.564} C_VEL
LIN {X 0,Y 316.045,Z 526.81,A -85,B 0,C 180,E1 14155.534,E2 14155.534} C_VEL
LIN {X 0,Y 315.754,Z 526.81,A -85,B 0,C 180,E1 14161.826,E2 14161.826} C_VEL
LIN {X 0,Y 315.48,Z 526.81,A -85,B 0,C 180,E1 14169.826,E2 14169.826} C_VEL
LIN {X 0,Y 315.5,Z 526.81,A -85,B 0,C 180,E1 14177.781,E2 14177.781} C_VEL
LIN {X 0,Y 315.633,Z 526.81,A -85,B 0,C 180,E1 14184.848,E2 14184.848} C_VEL
LIN {X 0,Y 315.879,Z 526.81,A -85,B 0,C 180,E1 14191.351,E2 14191.351} C_VEL
LIN {X 0,Y 316.164,Z 526.81,A -85,B 0,C 180,E1 14197.466,E2 14197.466} C_VEL
LIN {X 0,Y 316.507,Z 526.81,A -85,B 0,C 180,E1 14203.312,E2 14203.312} C_VEL
LIN {X 0,Y 317.004,Z 526.81,A -85,B 0,C 180,E1 14211.754,E2 14211.754} C_VEL
LIN {X 0,Y 317.656,Z 526.81,A -85,B 0,C 180,E1 14219.992,E2 14219.992} C_VEL
LIN {X 0,Y 316.982,Z 526.81,A -85,B 0,C 180,E1 14228.23,E2 14228.23} C_VEL
LIN {X 0,Y 316.494,Z 526.81,A -85,B 0,C 180,E1 14236.671,E2 14236.671} C_VEL
LIN {X 0,Y 316.06,Z 526.81,A -85,B 0,C 180,E1 14244.485,E2 14244.485} C_VEL
LIN {X 0,Y 315.798,Z 526.81,A -85,B 0,C 180,E1 14251.817,E2 14251.817} C_VEL
LIN {X 0,Y 315.467,Z 526.81,A -85,B 0,C 180,E1 14259.844,E2 14259.844} C_VEL
LIN {X 0,Y 315.39,Z 526.81,A -85,B 0,C 180,E1 14267.78,E2 14267.78} C_VEL
LIN {X 0,Y 315.835,Z 526.81,A -85,B 0,C 180,E1 14275.082,E2 14275.082} C_VEL
LIN {X 0,Y 334.466,Z 589.754,A -85,B 0,C 180,E1 14278.091,E2 14278.091} C_VEL
LIN {X 0,Y 331.33,Z 623.945,A -85,B 0,C 180,E1 14279.939,E2 14279.939} C_VEL
LIN {X 0,Y 327.52,Z 656.186,A -85,B 0,C 180,E1 14282.845,E2 14282.845} C_VEL
LIN {X 0,Y 323.797,Z 684.009,A -85,B 0,C 180,E1 14286.588,E2 14286.588} C_VEL
LIN {X 0,Y 320.964,Z 707.333,A -85,B 0,C 180,E1 14291.083,E2 14291.083} C_VEL
LIN {X 0,Y 319.516,Z 726.053,A -85,B 0,C 180,E1 14296.301,E2 14296.301} C_VEL
LIN {X 0,Y 319.466,Z 738.822,A -85,B 0,C 180,E1 14301.832,E2 14301.832} C_VEL
LIN {X 0,Y 319.712,Z 744.285,A -85,B 0,C 180,E1 14305.933,E2 14305.933} C_VEL
LIN {X 0,Y 319.968,Z 746.517,A -85,B 0,C 180,E1 14310.006,E2 14310.006} C_VEL
LIN {X 0,Y 319.407,Z 744.481,A -85,B 0,C 180,E1 14315.584,E2 14315.584} C_VEL
LIN {X 0,Y 318.973,Z 737.383,A -85,B 0,C 180,E1 14320.952,E2 14320.952} C_VEL
LIN {X 0,Y 319.906,Z 724.8,A -85,B 0,C 180,E1 14326.504,E2 14326.504} C_VEL
LIN {X 0,Y 322.961,Z 706.125,A -85,B 0,C 180,E1 14332.034,E2 14332.034} C_VEL
LIN {X 0,Y 328.429,Z 682.271,A -85,B 0,C 180,E1 14336.946,E2 14336.946} C_VEL
LIN {X 0,Y 335.462,Z 653.349,A -85,B 0,C 180,E1 14341.096,E2 14341.096} C_VEL
LIN {X 0,Y 342.969,Z 620.226,A -85,B 0,C 180,E1 14344.261,E2 14344.261} C_VEL
LIN {X 0,Y 345.86,Z 605.633,A -85,B 0,C 180,E1 14345.266,E2 14345.266} C_VEL
LIN {X 0,Y 345.414,Z 598.195,A -85,B 0,C 180,E1 14346.014,E2 14346.014} C_VEL
LIN {X 0,Y 341.639,Z 587.288,A -85,B 0,C 180,E1 14347.666,E2 14347.666} C_VEL
LIN {X 0,Y 335.94,Z 570.703,A -85,B 0,C 180,E1 14350.49,E2 14350.49} C_VEL
LIN {X 0,Y 330.086,Z 559.862,A -85,B 0,C 180,E1 14353.661,E2 14353.661} C_VEL
LIN {X 0,Y 327.424,Z 555.179,A -85,B 0,C 180,E1 14355.775,E2 14355.775} C_VEL
LIN {X 0,Y 325.132,Z 550.51,A -85,B 0,C 180,E1 14360.257,E2 14360.257} C_VEL
LIN {X 0,Y 327.052,Z 555.223,A -85,B 0,C 180,E1 14365.392,E2 14365.392} C_VEL
LIN {X 0,Y 331.515,Z 565.44,A -85,B 0,C 180,E1 14369.44,E2 14369.44} C_VEL
LIN {X 0,Y 335.638,Z 581.737,A -85,B 0,C 180,E1 14373.196,E2 14373.196} C_VEL
LIN {X 0,Y 335.83,Z 594.603,A -85,B 0,C 180,E1 14375.324,E2 14375.324} C_VEL
LIN {X 0,Y 329.423,Z 618.88,A -85,B 0,C 180,E1 14378.79,E2 14378.79} C_VEL
LIN {X 0,Y 323.397,Z 638.121,A -85,B 0,C 180,E1 14382.995,E2 14382.995} C_VEL
LIN {X 0,Y 318.937,Z 650.274,A -85,B 0,C 180,E1 14387.228,E2 14387.228} C_VEL
LIN {X 0,Y 315.643,Z 657.329,A -85,B 0,C 180,E1 14391.735,E2 14391.735} C_VEL
LIN {X 0,Y 314.393,Z 659.037,A -85,B 0,C 180,E1 14394.482,E2 14394.482} C_VEL
LIN {X 0,Y 313.419,Z 658.922,A -85,B 0,C 180,E1 14397.24,E2 14397.24} C_VEL
LIN {X 0,Y 312.443,Z 654.345,A -85,B 0,C 180,E1 14402.091,E2 14402.091} C_VEL
LIN {X 0,Y 312.664,Z 643.904,A -85,B 0,C 180,E1 14406.856,E2 14406.856} C_VEL
LIN {X 0,Y 313.65,Z 628.684,A -85,B 0,C 180,E1 14411.141,E2 14411.141} C_VEL
LIN {X 0,Y 315.461,Z 607.278,A -85,B 0,C 180,E1 14415.136,E2 14415.136} C_VEL
LIN {X 0,Y 317.566,Z 581.013,A -85,B 0,C 180,E1 14418.42,E2 14418.42} C_VEL
LIN {X 0,Y 317.025,Z 567.641,A -85,B 0,C 180,E1 14419.699,E2 14419.699} C_VEL
LIN {X 0,Y 310.853,Z 537.516,A -85,B 0,C 180,E1 14421.976,E2 14421.976} C_VEL
LIN {X 0,Y 308.378,Z 526.81,A -85,B 0,C 180,E1 14422.63,E2 14422.63} C_VEL
LIN {X 0,Y 307.894,Z 526.81,A -85,B 0,C 180,E1 14429.464,E2 14429.464} C_VEL
LIN {X 0,Y 307.573,Z 526.81,A -85,B 0,C 180,E1 14438.025,E2 14438.025} C_VEL
LIN {X 0,Y 307.59,Z 526.81,A -85,B 0,C 180,E1 14443.57,E2 14443.57} C_VEL
LIN {X 0,Y 307.654,Z 526.81,A -85,B 0,C 180,E1 14450.216,E2 14450.216} C_VEL
LIN {X 0,Y 307.751,Z 526.81,A -85,B 0,C 180,E1 14457.228,E2 14457.228} C_VEL
LIN {X 0,Y 308.054,Z 526.81,A -85,B 0,C 180,E1 14463.739,E2 14463.739} C_VEL
LIN {X 0,Y 308.371,Z 526.81,A -85,B 0,C 180,E1 14469.891,E2 14469.891} C_VEL
LIN {X 0,Y 308.614,Z 526.81,A -85,B 0,C 180,E1 14475.794,E2 14475.794} C_VEL
LIN {X 0,Y 309.285,Z 526.81,A -85,B 0,C 180,E1 14484.375,E2 14484.375} C_VEL
LIN {X 0,Y 309.801,Z 526.81,A -85,B 0,C 180,E1 14489.993,E2 14489.993} C_VEL
LIN {X 0,Y 309.075,Z 526.81,A -85,B 0,C 180,E1 14498.444,E2 14498.444} C_VEL
LIN {X 0,Y 308.593,Z 526.81,A -85,B 0,C 180,E1 14507.113,E2 14507.113} C_VEL
LIN {X 0,Y 308.209,Z 526.81,A -85,B 0,C 180,E1 14513.134,E2 14513.134} C_VEL
LIN {X 0,Y 307.894,Z 526.81,A -85,B 0,C 180,E1 14519.448,E2 14519.448} C_VEL
LIN {X 0,Y 307.559,Z 526.81,A -85,B 0,C 180,E1 14528.023,E2 14528.023} C_VEL
LIN {X 0,Y 307.555,Z 526.81,A -85,B 0,C 180,E1 14533.558,E2 14533.558} C_VEL
LIN {X 0,Y 307.627,Z 526.81,A -85,B 0,C 180,E1 14540.212,E2 14540.212} C_VEL
LIN {X 0,Y 307.722,Z 526.81,A -85,B 0,C 180,E1 14547.224,E2 14547.224} C_VEL
LIN {X 0,Y 308.029,Z 526.81,A -85,B 0,C 180,E1 14553.736,E2 14553.736} C_VEL
LIN {X 0,Y 308.376,Z 526.81,A -85,B 0,C 180,E1 14559.89,E2 14559.89} C_VEL
LIN {X 0,Y 308.655,Z 526.81,A -85,B 0,C 180,E1 14565.794,E2 14565.794} C_VEL
LIN {X 0,Y 309.3,Z 526.81,A -85,B 0,C 180,E1 14574.373,E2 14574.373} C_VEL
LIN {X 0,Y 309.753,Z 526.81,A -85,B 0,C 180,E1 14579.991,E2 14579.991} C_VEL
LIN {X 0,Y 309.038,Z 526.81,A -85,B 0,C 180,E1 14588.443,E2 14588.443} C_VEL
LIN {X 0,Y 308.547,Z 526.81,A -85,B 0,C 180,E1 14597.113,E2 14597.113} C_VEL
LIN {X 0,Y 308.174,Z 526.81,A -85,B 0,C 180,E1 14603.133,E2 14603.133} C_VEL
LIN {X 0,Y 307.909,Z 526.81,A -85,B 0,C 180,E1 14609.442,E2 14609.442} C_VEL
LIN {X 0,Y 307.615,Z 526.81,A -85,B 0,C 180,E1 14616.189,E2 14616.189} C_VEL
LIN {X 0,Y 307.491,Z 526.81,A -85,B 0,C 180,E1 14623.564,E2 14623.564} C_VEL
LIN {X 0,Y 307.524,Z 526.81,A -85,B 0,C 180,E1 14630.214,E2 14630.214} C_VEL
LIN {X 0,Y 307.82,Z 526.81,A -85,B 0,C 180,E1 14634.598,E2 14634.598} C_VEL
LIN {X 0,Y 326.759,Z 591.507,A -85,B 0,C 180,E1 14637.784,E2 14637.784} C_VEL
LIN {X 0,Y 323.472,Z 625.362,A -85,B 0,C 180,E1 14639.736,E2 14639.736} C_VEL
LIN {X 0,Y 319.637,Z 656.656,A -85,B 0,C 180,E1 14642.692,E2 14642.692} C_VEL
LIN {X 0,Y 315.878,Z 684.127,A -85,B 0,C 180,E1 14646.53,E2 14646.53} C_VEL
LIN {X 0,Y 312.985,Z 707.899,A -85,B 0,C 180,E1 14651.315,E2 14651.315} C_VEL
LIN {X 0,Y 311.695,Z 724.887,A -85,B 0,C 180,E1 14656.241,E2 14656.241} C_VEL
LIN {X 0,Y 311.628,Z 737.172,A -85,B 0,C 180,E1 14661.626,E2 14661.626} C_VEL
LIN {X 0,Y 311.919,Z 742.859,A -85,B 0,C 180,E1 14665.846,E2 14665.846} C_VEL
LIN {X 0,Y 312.172,Z 745.184,A -85,B 0,C 180,E1 14670.007,E2 14670.007} C_VEL
LIN {X 0,Y 311.58,Z 743.467,A -85,B 0,C 180,E1 14675.584,E2 14675.584} C_VEL
LIN {X 0,Y 311.092,Z 736.369,A -85,B 0,C 180,E1 14681.233,E2 14681.233} C_VEL
LIN {X 0,Y 312.153,Z 724.029,A -85,B 0,C 180,E1 14686.926,E2 14686.926} C_VEL
LIN {X 0,Y 315.826,Z 704.286,A -85,B 0,C 180,E1 14692.931,E2 14692.931} C_VEL
LIN {X 0,Y 321.969,Z 679.699,A -85,B 0,C 180,E1 14698.058,E2 14698.058} C_VEL
LIN {X 0,Y 329.476,Z 651.653,A -85,B 0,C 180,E1 14702.107,E2 14702.107} C_VEL
LIN {X 0,Y 337.084,Z 620.728,A -85,B 0,C 180,E1 14705.142,E2 14705.142} C_VEL
LIN {X 0,Y 342.596,Z 592.241,A -85,B 0,C 180,E1 14707.04,E2 14707.04} C_VEL
LIN {X 0,Y 341.639,Z 587.288,A -85,B 0,C 180,E1 14707.666,E2 14707.666} C_VEL
LIN {X 0,Y 337.529,Z 579.56,A -85,B 0,C 180,E1 14709.299,E2 14709.299} C_VEL
LIN {X 0,Y 329.4,Z 570.968,A -85,B 0,C 180,E1 14712.611,E2 14712.611} C_VEL
LIN {X 0,Y 324.969,Z 562.51,A -85,B 0,C 180,E1 14716.062,E2 14716.062} C_VEL
LIN {X 0,Y 322.996,Z 558.107,A -85,B 0,C 180,E1 14719.942,E2 14719.942} C_VEL
LIN {X 0,Y 324,Z 562.277,A -85,B 0,C 180,E1 14724.924,E2 14724.924} C_VEL
LIN {X 0,Y 327.601,Z 572.011,A -85,B 0,C 180,E1 14729.066,E2 14729.066} C_VEL
LIN {X 0,Y 330.488,Z 587.273,A -85,B 0,C 180,E1 14732.744,E2 14732.744} C_VEL
LIN {X 0,Y 329.993,Z 598.142,A -85,B 0,C 180,E1 14734.59,E2 14734.59} C_VEL
LIN {X 0,Y 322.724,Z 622.718,A -85,B 0,C 180,E1 14738.328,E2 14738.328} C_VEL
LIN {X 0,Y 316.303,Z 641.011,A -85,B 0,C 180,E1 14742.602,E2 14742.602} C_VEL
LIN {X 0,Y 311.58,Z 652.5,A -85,B 0,C 180,E1 14746.896,E2 14746.896} C_VEL
LIN {X 0,Y 308.052,Z 659.098,A -85,B 0,C 180,E1 14751.53,E2 14751.53} C_VEL
LIN {X 0,Y 306.693,Z 660.522,A -85,B 0,C 180,E1 14754.343,E2 14754.343} C_VEL
LIN {X 0,Y 305.193,Z 659.365,A -85,B 0,C 180,E1 14758.587,E2 14758.587} C_VEL
LIN {X 0,Y 304.584,Z 652.639,A -85,B 0,C 180,E1 14763.571,E2 14763.571} C_VEL
LIN {X 0,Y 305.039,Z 640.778,A -85,B 0,C 180,E1 14768.212,E2 14768.212} C_VEL
LIN {X 0,Y 306.429,Z 621.931,A -85,B 0,C 180,E1 14772.855,E2 14772.855} C_VEL
LIN {X 0,Y 308.53,Z 598.222,A -85,B 0,C 180,E1 14776.73,E2 14776.73} C_VEL
LIN {X 0,Y 309.971,Z 573.013,A -85,B 0,C 180,E1 14779.537,E2 14779.537} C_VEL
LIN {X 0,Y 304.22,Z 543.311,A -85,B 0,C 180,E1 14781.993,E2 14781.993} C_VEL
LIN {X 0,Y 300.443,Z 526.81,A -85,B 0,C 180,E1 14783,E2 14783} C_VEL
LIN {X 0,Y 299.799,Z 526.81,A -85,B 0,C 180,E1 14790.833,E2 14790.833} C_VEL
LIN {X 0,Y 299.673,Z 526.81,A -85,B 0,C 180,E1 14797.331,E2 14797.331} C_VEL
LIN {X 0,Y 299.609,Z 526.81,A -85,B 0,C 180,E1 14805.04,E2 14805.04} C_VEL
LIN {X 0,Y 299.712,Z 526.81,A -85,B 0,C 180,E1 14812.676,E2 14812.676} C_VEL
LIN {X 0,Y 299.886,Z 526.81,A -85,B 0,C 180,E1 14819.669,E2 14819.669} C_VEL
LIN {X 0,Y 300.209,Z 526.81,A -85,B 0,C 180,E1 14826.197,E2 14826.197} C_VEL
LIN {X 0,Y 300.619,Z 526.81,A -85,B 0,C 180,E1 14833.145,E2 14833.145} C_VEL
LIN {X 0,Y 301.11,Z 526.81,A -85,B 0,C 180,E1 14841.317,E2 14841.317} C_VEL
LIN {X 0,Y 301.716,Z 526.81,A -85,B 0,C 180,E1 14847.117,E2 14847.117} C_VEL
LIN {X 0,Y 301.688,Z 526.81,A -85,B 0,C 180,E1 14852.87,E2 14852.87} C_VEL
LIN {X 0,Y 300.989,Z 526.81,A -85,B 0,C 180,E1 14861.601,E2 14861.601} C_VEL
LIN {X 0,Y 300.604,Z 526.81,A -85,B 0,C 180,E1 14867.583,E2 14867.583} C_VEL
LIN {X 0,Y 300.117,Z 526.81,A -85,B 0,C 180,E1 14874.743,E2 14874.743} C_VEL
LIN {X 0,Y 299.8,Z 526.81,A -85,B 0,C 180,E1 14880.834,E2 14880.834} C_VEL
LIN {X 0,Y 299.659,Z 526.81,A -85,B 0,C 180,E1 14887.315,E2 14887.315} C_VEL
LIN {X 0,Y 299.594,Z 526.81,A -85,B 0,C 180,E1 14895.024,E2 14895.024} C_VEL
LIN {X 0,Y 299.681,Z 526.81,A -85,B 0,C 180,E1 14902.671,E2 14902.671} C_VEL
LIN {X 0,Y 299.858,Z 526.81,A -85,B 0,C 180,E1 14909.665,E2 14909.665} C_VEL
LIN {X 0,Y 300.186,Z 526.81,A -85,B 0,C 180,E1 14916.194,E2 14916.194} C_VEL
LIN {X 0,Y 300.661,Z 526.81,A -85,B 0,C 180,E1 14923.074,E2 14923.074} C_VEL
LIN {X 0,Y 301.107,Z 526.81,A -85,B 0,C 180,E1 14931.744,E2 14931.744} C_VEL
LIN {X 0,Y 301.859,Z 526.81,A -85,B 0,C 180,E1 14939.991,E2 14939.991} C_VEL
LIN {X 0,Y 301.372,Z 526.81,A -85,B 0,C 180,E1 14945.758,E2 14945.758} C_VEL
LIN {X 0,Y 300.725,Z 526.81,A -85,B 0,C 180,E1 14954.57,E2 14954.57} C_VEL
LIN {X 0,Y 300.38,Z 526.81,A -85,B 0,C 180,E1 14960.65,E2 14960.65} C_VEL
LIN {X 0,Y 300.059,Z 526.81,A -85,B 0,C 180,E1 14966.998,E2 14966.998} C_VEL
LIN {X 0,Y 299.768,Z 526.81,A -85,B 0,C 180,E1 14973.739,E2 14973.739} C_VEL
LIN {X 0,Y 299.577,Z 526.81,A -85,B 0,C 180,E1 14981.059,E2 14981.059} C_VEL
LIN {X 0,Y 299.553,Z 526.81,A -85,B 0,C 180,E1 14989.285,E2 14989.285} C_VEL
LIN {X 0,Y 299.847,Z 527.063,A -85,B 0,C 180,E1 14994.122,E2 14994.122} C_VEL
LIN {X 0,Y 319.164,Z 591.853,A -85,B 0,C 180,E1 14997.421,E2 14997.421} C_VEL
LIN {X 0,Y 315.752,Z 625.468,A -85,B 0,C 180,E1 14999.438,E2 14999.438} C_VEL
LIN {X 0,Y 311.769,Z 657.002,A -85,B 0,C 180,E1 15002.533,E2 15002.533} C_VEL
LIN {X 0,Y 307.93,Z 684.552,A -85,B 0,C 180,E1 15006.547,E2 15006.547} C_VEL
LIN {X 0,Y 305.05,Z 707.89,A -85,B 0,C 180,E1 15011.452,E2 15011.452} C_VEL
LIN {X 0,Y 303.816,Z 725.283,A -85,B 0,C 180,E1 15016.76,E2 15016.76} C_VEL
LIN {X 0,Y 303.888,Z 736.678,A -85,B 0,C 180,E1 15022.132,E2 15022.132} C_VEL
LIN {X 0,Y 304.228,Z 742.514,A -85,B 0,C 180,E1 15027.154,E2 15027.154} C_VEL
LIN {X 0,Y 304.405,Z 743.842,A -85,B 0,C 180,E1 15030.007,E2 15030.007} C_VEL
LIN {X 0,Y 303.718,Z 742.284,A -85,B 0,C 180,E1 15035.729,E2 15035.729} C_VEL
LIN {X 0,Y 303.239,Z 735.381,A -85,B 0,C 180,E1 15041.527,E2 15041.527} C_VEL
LIN {X 0,Y 304.652,Z 721.721,A -85,B 0,C 180,E1 15047.954,E2 15047.954} C_VEL
LIN {X 0,Y 308.715,Z 702.688,A -85,B 0,C 180,E1 15053.834,E2 15053.834} C_VEL
LIN {X 0,Y 315.492,Z 678.043,A -85,B 0,C 180,E1 15059.079,E2 15059.079} C_VEL
LIN {X 0,Y 323.607,Z 650.25,A -85,B 0,C 180,E1 15063.156,E2 15063.156} C_VEL
LIN {X 0,Y 332.172,Z 617.866,A -85,B 0,C 180,E1 15066.346,E2 15066.346} C_VEL
LIN {X 0,Y 336.978,Z 594.222,A -85,B 0,C 180,E1 15068.019,E2 15068.019} C_VEL
LIN {X 0,Y 332.751,Z 578.596,A -85,B 0,C 180,E1 15070.657,E2 15070.657} C_VEL
LIN {X 0,Y 329.4,Z 570.968,A -85,B 0,C 180,E1 15072.611,E2 15072.611} C_VEL
LIN {X 0,Y 325.651,Z 567.892,A -85,B 0,C 180,E1 15074.737,E2 15074.737} C_VEL
LIN {X 0,Y 320.78,Z 567.168,A -85,B 0,C 180,E1 15078.625,E2 15078.625} C_VEL
LIN {X 0,Y 320.442,Z 565.755,A -85,B 0,C 180,E1 15080.756,E2 15080.756} C_VEL
LIN {X 0,Y 321.564,Z 570.93,A -85,B 0,C 180,E1 15085.609,E2 15085.609} C_VEL
LIN {X 0,Y 324.193,Z 581.481,A -85,B 0,C 180,E1 15089.573,E2 15089.573} C_VEL
LIN {X 0,Y 325.257,Z 595.662,A -85,B 0,C 180,E1 15092.838,E2 15092.838} C_VEL
LIN {X 0,Y 323.027,Z 605.814,A -85,B 0,C 180,E1 15094.368,E2 15094.368} C_VEL
LIN {X 0,Y 315.457,Z 628.192,A -85,B 0,C 180,E1 15098.173,E2 15098.173} C_VEL
LIN {X 0,Y 308.789,Z 644.969,A -85,B 0,C 180,E1 15102.533,E2 15102.533} C_VEL
LIN {X 0,Y 303.411,Z 656.387,A -85,B 0,C 180,E1 15107.518,E2 15107.518} C_VEL
LIN {X 0,Y 300.456,Z 660.837,A -85,B 0,C 180,E1 15111.314,E2 15111.314} C_VEL
LIN {X 0,Y 298.975,Z 662.016,A -85,B 0,C 180,E1 15114.196,E2 15114.196} C_VEL
LIN {X 0,Y 297.371,Z 660.448,A -85,B 0,C 180,E1 15118.55,E2 15118.55} C_VEL
LIN {X 0,Y 296.728,Z 653.328,A -85,B 0,C 180,E1 15123.664,E2 15123.664} C_VEL
LIN {X 0,Y 297.271,Z 639.793,A -85,B 0,C 180,E1 15128.798,E2 15128.798} C_VEL
LIN {X 0,Y 298.689,Z 621.618,A -85,B 0,C 180,E1 15133.194,E2 15133.194} C_VEL
LIN {X 0,Y 300.766,Z 598.404,A -85,B 0,C 180,E1 15137.005,E2 15137.005} C_VEL
LIN {X 0,Y 302.059,Z 572.956,A -85,B 0,C 180,E1 15139.88,E2 15139.88} C_VEL
LIN {X 0,Y 296.046,Z 542.57,A -85,B 0,C 180,E1 15142.429,E2 15142.429} C_VEL
LIN {X 0,Y 292.437,Z 526.81,A -85,B 0,C 180,E1 15143.446,E2 15143.446} C_VEL
LIN {X 0,Y 291.843,Z 526.81,A -85,B 0,C 180,E1 15151.26,E2 15151.26} C_VEL
LIN {X 0,Y 291.638,Z 526.81,A -85,B 0,C 180,E1 15158.844,E2 15158.844} C_VEL
LIN {X 0,Y 291.59,Z 526.81,A -85,B 0,C 180,E1 15167.535,E2 15167.535} C_VEL
LIN {X 0,Y 291.859,Z 526.81,A -85,B 0,C 180,E1 15176.113,E2 15176.113} C_VEL
LIN {X 0,Y 292.057,Z 526.81,A -85,B 0,C 180,E1 15182.18,E2 15182.18} C_VEL
LIN {X 0,Y 292.426,Z 526.81,A -85,B 0,C 180,E1 15188.761,E2 15188.761} C_VEL
LIN {X 0,Y 292.747,Z 526.81,A -85,B 0,C 180,E1 15195.006,E2 15195.006} C_VEL
LIN {X 0,Y 293.156,Z 526.81,A -85,B 0,C 180,E1 15201.08,E2 15201.08} C_VEL
LIN {X 0,Y 293.789,Z 526.81,A -85,B 0,C 180,E1 15207.039,E2 15207.039} C_VEL
LIN {X 0,Y 293.764,Z 526.81,A -85,B 0,C 180,E1 15212.947,E2 15212.947} C_VEL
LIN {X 0,Y 293.042,Z 526.81,A -85,B 0,C 180,E1 15221.92,E2 15221.92} C_VEL
LIN {X 0,Y 292.614,Z 526.81,A -85,B 0,C 180,E1 15228.079,E2 15228.079} C_VEL
LIN {X 0,Y 292.232,Z 526.81,A -85,B 0,C 180,E1 15234.479,E2 15234.479} C_VEL
LIN {X 0,Y 291.869,Z 526.81,A -85,B 0,C 180,E1 15241.24,E2 15241.24} C_VEL
LIN {X 0,Y 291.616,Z 526.81,A -85,B 0,C 180,E1 15248.838,E2 15248.838} C_VEL
LIN {X 0,Y 291.562,Z 526.81,A -85,B 0,C 180,E1 15257.53,E2 15257.53} C_VEL
LIN {X 0,Y 291.826,Z 526.81,A -85,B 0,C 180,E1 15266.098,E2 15266.098} C_VEL
LIN {X 0,Y 292.029,Z 526.81,A -85,B 0,C 180,E1 15272.176,E2 15272.176} C_VEL
LIN {X 0,Y 292.396,Z 526.81,A -85,B 0,C 180,E1 15278.739,E2 15278.739} C_VEL
LIN {X 0,Y 292.779,Z 526.81,A -85,B 0,C 180,E1 15285.006,E2 15285.006} C_VEL
LIN {X 0,Y 293.158,Z 526.81,A -85,B 0,C 180,E1 15291.749,E2 15291.749} C_VEL
LIN {X 0,Y 293.954,Z 526.81,A -85,B 0,C 180,E1 15299.991,E2 15299.991} C_VEL
LIN {X 0,Y 293.433,Z 526.81,A -85,B 0,C 180,E1 15305.914,E2 15305.914} C_VEL
LIN {X 0,Y 292.979,Z 526.81,A -85,B 0,C 180,E1 15311.92,E2 15311.92} C_VEL
LIN {X 0,Y 292.568,Z 526.81,A -85,B 0,C 180,E1 15318.079,E2 15318.079} C_VEL
LIN {X 0,Y 292.204,Z 526.81,A -85,B 0,C 180,E1 15324.478,E2 15324.478} C_VEL
LIN {X 0,Y 291.918,Z 526.81,A -85,B 0,C 180,E1 15331.23,E2 15331.23} C_VEL
LIN {X 0,Y 291.603,Z 526.81,A -85,B 0,C 180,E1 15338.857,E2 15338.857} C_VEL
LIN {X 0,Y 291.468,Z 526.81,A -85,B 0,C 180,E1 15347.532,E2 15347.532} C_VEL
LIN {X 0,Y 291.864,Z 527.211,A -85,B 0,C 180,E1 15353.616,E2 15353.616} C_VEL
LIN {X 0,Y 311.485,Z 592.716,A -85,B 0,C 180,E1 15357.075,E2 15357.075} C_VEL
LIN {X 0,Y 307.995,Z 625.941,A -85,B 0,C 180,E1 15359.169,E2 15359.169} C_VEL
LIN {X 0,Y 303.907,Z 657.23,A -85,B 0,C 180,E1 15362.365,E2 15362.365} C_VEL
LIN {X 0,Y 299.955,Z 684.988,A -85,B 0,C 180,E1 15366.585,E2 15366.585} C_VEL
LIN {X 0,Y 297.11,Z 707.923,A -85,B 0,C 180,E1 15371.632,E2 15371.632} C_VEL
LIN {X 0,Y 295.981,Z 725.34,A -85,B 0,C 180,E1 15377.247,E2 15377.247} C_VEL
LIN {X 0,Y 296.163,Z 736.136,A -85,B 0,C 180,E1 15382.664,E2 15382.664} C_VEL
LIN {X 0,Y 296.46,Z 741.031,A -85,B 0,C 180,E1 15387.079,E2 15387.079} C_VEL
LIN {X 0,Y 296.612,Z 742.484,A -85,B 0,C 180,E1 15390.007,E2 15390.007} C_VEL
LIN {X 0,Y 295.856,Z 741.076,A -85,B 0,C 180,E1 15395.882,E2 15395.882} C_VEL
LIN {X 0,Y 295.362,Z 734.413,A -85,B 0,C 180,E1 15401.839,E2 15401.839} C_VEL
LIN {X 0,Y 296.937,Z 721.184,A -85,B 0,C 180,E1 15408.381,E2 15408.381} C_VEL
LIN {X 0,Y 301.576,Z 701.833,A -85,B 0,C 180,E1 15414.606,E2 15414.606} C_VEL
LIN {X 0,Y 309.115,Z 676.721,A -85,B 0,C 180,E1 15420.112,E2 15420.112} C_VEL
LIN {X 0,Y 317.92,Z 649.071,A -85,B 0,C 180,E1 15424.241,E2 15424.241} C_VEL
LIN {X 0,Y 327.364,Z 616.126,A -85,B 0,C 180,E1 15427.524,E2 15427.524} C_VEL
LIN {X 0,Y 331.666,Z 597.158,A -85,B 0,C 180,E1 15428.915,E2 15428.915} C_VEL
LIN {X 0,Y 327.934,Z 582.317,A -85,B 0,C 180,E1 15431.733,E2 15431.733} C_VEL
LIN {X 0,Y 322.987,Z 570.531,A -85,B 0,C 180,E1 15435.722,E2 15435.722} C_VEL
LIN {X 0,Y 320.78,Z 567.168,A -85,B 0,C 180,E1 15438.625,E2 15438.625} C_VEL
LIN {X 0,Y 319.987,Z 567.368,A -85,B 0,C 180,E1 15440.165,E2 15440.165} C_VEL
LIN {X 0,Y 317.952,Z 577.055,A -85,B 0,C 180,E1 15444.701,E2 15444.701} C_VEL
LIN {X 0,Y 319.639,Z 585.898,A -85,B 0,C 180,E1 15448.609,E2 15448.609} C_VEL
LIN {X 0,Y 320.001,Z 599.62,A -85,B 0,C 180,E1 15452.064,E2 15452.064} C_VEL
LIN {X 0,Y 316.335,Z 612.334,A -85,B 0,C 180,E1 15454.022,E2 15454.022} C_VEL
LIN {X 0,Y 308.222,Z 633.448,A -85,B 0,C 180,E1 15458.013,E2 15458.013} C_VEL
LIN {X 0,Y 300.752,Z 649.847,A -85,B 0,C 180,E1 15462.845,E2 15462.845} C_VEL
LIN {X 0,Y 295.179,Z 659.862,A -85,B 0,C 180,E1 15468.17,E2 15468.17} C_VEL
LIN {X 0,Y 292.842,Z 662.58,A -85,B 0,C 180,E1 15471.087,E2 15471.087} C_VEL
LIN {X 0,Y 291.281,Z 663.516,A -85,B 0,C 180,E1 15474.042,E2 15474.042} C_VEL
LIN {X 0,Y 289.562,Z 661.516,A -85,B 0,C 180,E1 15478.511,E2 15478.511} C_VEL
LIN {X 0,Y 288.88,Z 654.021,A -85,B 0,C 180,E1 15483.751,E2 15483.751} C_VEL
LIN {X 0,Y 289.455,Z 639.91,A -85,B 0,C 180,E1 15489.037,E2 15489.037} C_VEL
LIN {X 0,Y 290.945,Z 621.192,A -85,B 0,C 180,E1 15493.552,E2 15493.552} C_VEL
LIN {X 0,Y 293.156,Z 596.869,A -85,B 0,C 180,E1 15497.516,E2 15497.516} C_VEL
LIN {X 0,Y 294.439,Z 574.877,A -85,B 0,C 180,E1 15500.03,E2 15500.03} C_VEL
LIN {X 0,Y 288.664,Z 545.222,A -85,B 0,C 180,E1 15502.647,E2 15502.647} C_VEL
LIN {X 0,Y 284.491,Z 526.81,A -85,B 0,C 180,E1 15503.921,E2 15503.921} C_VEL
LIN {X 0,Y 283.873,Z 526.81,A -85,B 0,C 180,E1 15512.242,E2 15512.242} C_VEL
LIN {X 0,Y 283.607,Z 526.81,A -85,B 0,C 180,E1 15519.849,E2 15519.849} C_VEL
LIN {X 0,Y 283.604,Z 526.81,A -85,B 0,C 180,E1 15528.378,E2 15528.378} C_VEL
LIN {X 0,Y 283.736,Z 526.81,A -85,B 0,C 180,E1 15534.048,E2 15534.048} C_VEL
LIN {X 0,Y 284.065,Z 526.81,A -85,B 0,C 180,E1 15541.326,E2 15541.326} C_VEL
LIN {X 0,Y 284.413,Z 526.81,A -85,B 0,C 180,E1 15548.113,E2 15548.113} C_VEL
LIN {X 0,Y 284.769,Z 526.81,A -85,B 0,C 180,E1 15554.576,E2 15554.576} C_VEL
LIN {X 0,Y 285.213,Z 526.81,A -85,B 0,C 180,E1 15560.829,E2 15560.829} C_VEL
LIN {X 0,Y 285.88,Z 526.81,A -85,B 0,C 180,E1 15566.957,E2 15566.957} C_VEL
LIN {X 0,Y 285.862,Z 526.81,A -85,B 0,C 180,E1 15573.029,E2 15573.029} C_VEL
LIN {X 0,Y 285.074,Z 526.81,A -85,B 0,C 180,E1 15582.258,E2 15582.258} C_VEL
LIN {X 0,Y 284.649,Z 526.81,A -85,B 0,C 180,E1 15588.604,E2 15588.604} C_VEL
LIN {X 0,Y 284.212,Z 526.81,A -85,B 0,C 180,E1 15595.217,E2 15595.217} C_VEL
LIN {X 0,Y 283.88,Z 526.81,A -85,B 0,C 180,E1 15602.223,E2 15602.223} C_VEL
LIN {X 0,Y 283.581,Z 526.81,A -85,B 0,C 180,E1 15609.834,E2 15609.834} C_VEL
LIN {X 0,Y 283.577,Z 526.81,A -85,B 0,C 180,E1 15618.362,E2 15618.362} C_VEL
LIN {X 0,Y 283.704,Z 526.81,A -85,B 0,C 180,E1 15624.043,E2 15624.043} C_VEL
LIN {X 0,Y 284.035,Z 526.81,A -85,B 0,C 180,E1 15631.322,E2 15631.322} C_VEL
LIN {X 0,Y 284.389,Z 526.81,A -85,B 0,C 180,E1 15638.11,E2 15638.11} C_VEL
LIN {X 0,Y 284.798,Z 526.81,A -85,B 0,C 180,E1 15644.576,E2 15644.576} C_VEL
LIN {X 0,Y 285.22,Z 526.81,A -85,B 0,C 180,E1 15651.759,E2 15651.759} C_VEL
LIN {X 0,Y 286.079,Z 526.81,A -85,B 0,C 180,E1 15659.991,E2 15659.991} C_VEL
LIN {X 0,Y 285.491,Z 526.81,A -85,B 0,C 180,E1 15666.079,E2 15666.079} C_VEL
LIN {X 0,Y 285.015,Z 526.81,A -85,B 0,C 180,E1 15672.258,E2 15672.258} C_VEL
LIN {X 0,Y 284.6,Z 526.81,A -85,B 0,C 180,E1 15678.604,E2 15678.604} C_VEL
LIN {X 0,Y 284.195,Z 526.81,A -85,B 0,C 180,E1 15685.215,E2 15685.215} C_VEL
LIN {X 0,Y 283.936,Z 526.81,A -85,B 0,C 180,E1 15692.212,E2 15692.212} C_VEL
LIN {X 0,Y 283.557,Z 526.81,A -85,B 0,C 180,E1 15699.833,E2 15699.833} C_VEL
LIN {X 0,Y 283.492,Z 526.81,A -85,B 0,C 180,E1 15708.375,E2 15708.375} C_VEL
LIN {X 0,Y 283.926,Z 527.149,A -85,B 0,C 180,E1 15713.1,E2 15713.1} C_VEL
LIN {X 0,Y 303.534,Z 592.529,A -85,B 0,C 180,E1 15716.667,E2 15716.667} C_VEL
LIN {X 0,Y 300.469,Z 624.393,A -85,B 0,C 180,E1 15718.739,E2 15718.739} C_VEL
LIN {X 0,Y 296.286,Z 655.853,A -85,B 0,C 180,E1 15722.006,E2 15722.006} C_VEL
LIN {X 0,Y 292.225,Z 683.746,A -85,B 0,C 180,E1 15726.333,E2 15726.333} C_VEL
LIN {X 0,Y 289.404,Z 705.882,A -85,B 0,C 180,E1 15731.275,E2 15731.275} C_VEL
LIN {X 0,Y 288.178,Z 723.268,A -85,B 0,C 180,E1 15736.896,E2 15736.896} C_VEL
LIN {X 0,Y 288.376,Z 734.377,A -85,B 0,C 180,E1 15742.465,E2 15742.465} C_VEL
LIN {X 0,Y 288.687,Z 739.519,A -85,B 0,C 180,E1 15747.001,E2 15747.001} C_VEL
LIN {X 0,Y 288.842,Z 741.117,A -85,B 0,C 180,E1 15750.007,E2 15750.007} C_VEL
LIN {X 0,Y 288,Z 739.869,A -85,B 0,C 180,E1 15756.043,E2 15756.043} C_VEL
LIN {X 0,Y 287.516,Z 733.43,A -85,B 0,C 180,E1 15762.167,E2 15762.167} C_VEL
LIN {X 0,Y 289.38,Z 719.959,A -85,B 0,C 180,E1 15769.111,E2 15769.111} C_VEL
LIN {X 0,Y 294.434,Z 701.105,A -85,B 0,C 180,E1 15775.405,E2 15775.405} C_VEL
LIN {X 0,Y 302.258,Z 677.316,A -85,B 0,C 180,E1 15780.85,E2 15780.85} C_VEL
LIN {X 0,Y 311.957,Z 649.427,A -85,B 0,C 180,E1 15785.202,E2 15785.202} C_VEL
LIN {X 0,Y 321.838,Z 618.078,A -85,B 0,C 180,E1 15788.475,E2 15788.475} C_VEL
LIN {X 0,Y 326.505,Z 600.604,A -85,B 0,C 180,E1 15789.794,E2 15789.794} C_VEL
LIN {X 0,Y 323.86,Z 588.206,A -85,B 0,C 180,E1 15792.325,E2 15792.325} C_VEL
LIN {X 0,Y 319.781,Z 577.378,A -85,B 0,C 180,E1 15796.26,E2 15796.26} C_VEL
LIN {X 0,Y 317.887,Z 573.761,A -85,B 0,C 180,E1 15799.657,E2 15799.657} C_VEL
LIN {X 0,Y 317.443,Z 575.247,A -85,B 0,C 180,E1 15803.057,E2 15803.057} C_VEL
LIN {X 0,Y 317.952,Z 577.055,A -85,B 0,C 180,E1 15804.701,E2 15804.701} C_VEL
LIN {X 0,Y 317.76,Z 583.171,A -85,B 0,C 180,E1 15806.784,E2 15806.784} C_VEL
LIN {X 0,Y 315.39,Z 597.913,A -85,B 0,C 180,E1 15809.869,E2 15809.869} C_VEL
LIN {X 0,Y 313.864,Z 607.651,A -85,B 0,C 180,E1 15811.955,E2 15811.955} C_VEL
LIN {X 0,Y 304.836,Z 629.948,A -85,B 0,C 180,E1 15815.821,E2 15815.821} C_VEL
LIN {X 0,Y 296.278,Z 647.828,A -85,B 0,C 180,E1 15820.61,E2 15820.61} C_VEL
LIN {X 0,Y 289.699,Z 659.139,A -85,B 0,C 180,E1 15825.748,E2 15825.748} C_VEL
LIN {X 0,Y 285.253,Z 664.35,A -85,B 0,C 180,E1 15830.848,E2 15830.848} C_VEL
LIN {X 0,Y 283.554,Z 664.943,A -85,B 0,C 180,E1 15833.879,E2 15833.879} C_VEL
LIN {X 0,Y 281.76,Z 662.579,A -85,B 0,C 180,E1 15838.47,E2 15838.47} C_VEL
LIN {X 0,Y 281.038,Z 654.541,A -85,B 0,C 180,E1 15843.856,E2 15843.856} C_VEL
LIN {X 0,Y 281.544,Z 641.254,A -85,B 0,C 180,E1 15848.903,E2 15848.903} C_VEL
LIN {X 0,Y 283.035,Z 622.523,A -85,B 0,C 180,E1 15853.544,E2 15853.544} C_VEL
LIN {X 0,Y 285.336,Z 597.779,A -85,B 0,C 180,E1 15857.698,E2 15857.698} C_VEL
LIN {X 0,Y 286.644,Z 575.629,A -85,B 0,C 180,E1 15860.308,E2 15860.308} C_VEL
LIN {X 0,Y 280.754,Z 545.416,A -85,B 0,C 180,E1 15863.026,E2 15863.026} C_VEL
LIN {X 0,Y 276.511,Z 526.81,A -85,B 0,C 180,E1 15864.282,E2 15864.282} C_VEL
LIN {X 0,Y 275.799,Z 526.81,A -85,B 0,C 180,E1 15873.306,E2 15873.306} C_VEL
LIN {X 0,Y 275.67,Z 526.81,A -85,B 0,C 180,E1 15881.24,E2 15881.24} C_VEL
LIN {X 0,Y 275.688,Z 526.81,A -85,B 0,C 180,E1 15888.764,E2 15888.764} C_VEL
LIN {X 0,Y 275.847,Z 526.81,A -85,B 0,C 180,E1 15896.701,E2 15896.701} C_VEL
LIN {X 0,Y 276.208,Z 526.81,A -85,B 0,C 180,E1 15903.982,E2 15903.982} C_VEL
LIN {X 0,Y 276.602,Z 526.81,A -85,B 0,C 180,E1 15910.819,E2 15910.819} C_VEL
LIN {X 0,Y 277.123,Z 526.81,A -85,B 0,C 180,E1 15919.594,E2 15919.594} C_VEL
LIN {X 0,Y 277.948,Z 526.81,A -85,B 0,C 180,E1 15926.87,E2 15926.87} C_VEL
LIN {X 0,Y 277.934,Z 526.81,A -85,B 0,C 180,E1 15933.115,E2 15933.115} C_VEL
LIN {X 0,Y 277.106,Z 526.81,A -85,B 0,C 180,E1 15942.617,E2 15942.617} C_VEL
LIN {X 0,Y 276.501,Z 526.81,A -85,B 0,C 180,E1 15951.408,E2 15951.408} C_VEL
LIN {X 0,Y 276.045,Z 526.81,A -85,B 0,C 180,E1 15959.571,E2 15959.571} C_VEL
LIN {X 0,Y 275.687,Z 526.81,A -85,B 0,C 180,E1 15967.156,E2 15967.156} C_VEL
LIN {X 0,Y 275.633,Z 526.81,A -85,B 0,C 180,E1 15975.559,E2 15975.559} C_VEL
LIN {X 0,Y 275.706,Z 526.81,A -85,B 0,C 180,E1 15982.828,E2 15982.828} C_VEL
LIN {X 0,Y 276.156,Z 526.81,A -85,B 0,C 180,E1 15991.294,E2 15991.294} C_VEL
LIN {X 0,Y 276.47,Z 526.81,A -85,B 0,C 180,E1 15998.57,E2 15998.57} C_VEL
LIN {X 0,Y 277.04,Z 526.81,A -85,B 0,C 180,E1 16007.364,E2 16007.364} C_VEL
LIN {X 0,Y 277.905,Z 526.81,A -85,B 0,C 180,E1 16016.867,E2 16016.867} C_VEL
LIN {X 0,Y 277.903,Z 526.81,A -85,B 0,C 180,E1 16023.113,E2 16023.113} C_VEL
LIN {X 0,Y 277.047,Z 526.81,A -85,B 0,C 180,E1 16032.616,E2 16032.616} C_VEL
LIN {X 0,Y 276.509,Z 526.81,A -85,B 0,C 180,E1 16041.451,E2 16041.451} C_VEL
LIN {X 0,Y 276.055,Z 526.81,A -85,B 0,C 180,E1 16049.566,E2 16049.566} C_VEL
LIN {X 0,Y 275.695,Z 526.81,A -85,B 0,C 180,E1 16057.15,E2 16057.15} C_VEL
LIN {X 0,Y 275.549,Z 526.81,A -85,B 0,C 180,E1 16065.57,E2 16065.57} C_VEL
LIN {X 0,Y 275.967,Z 526.81,A -85,B 0,C 180,E1 16072.529,E2 16072.529} C_VEL
LIN {X 0,Y 295.245,Z 592.133,A -85,B 0,C 180,E1 16076.226,E2 16076.226} C_VEL
LIN {X 0,Y 295.261,Z 603.951,A -85,B 0,C 180,E1 16076.935,E2 16076.935} C_VEL
LIN {X 0,Y 291.26,Z 636.392,A -85,B 0,C 180,E1 16079.555,E2 16079.555} C_VEL
LIN {X 0,Y 286.736,Z 666.638,A -85,B 0,C 180,E1 16083.354,E2 16083.354} C_VEL
LIN {X 0,Y 283.14,Z 691.993,A -85,B 0,C 180,E1 16088.026,E2 16088.026} C_VEL
LIN {X 0,Y 280.86,Z 712.827,A -85,B 0,C 180,E1 16093.567,E2 16093.567} C_VEL
LIN {X 0,Y 280.327,Z 726.942,A -85,B 0,C 180,E1 16099.111,E2 16099.111} C_VEL
LIN {X 0,Y 280.701,Z 734.77,A -85,B 0,C 180,E1 16103.814,E2 16103.814} C_VEL
LIN {X 0,Y 280.915,Z 737.985,A -85,B 0,C 180,E1 16106.918,E2 16106.918} C_VEL
LIN {X 0,Y 281.067,Z 739.681,A -85,B 0,C 180,E1 16110.007,E2 16110.007} C_VEL
LIN {X 0,Y 280.13,Z 738.661,A -85,B 0,C 180,E1 16116.213,E2 16116.213} C_VEL
LIN {X 0,Y 279.719,Z 731.672,A -85,B 0,C 180,E1 16123.071,E2 16123.071} C_VEL
LIN {X 0,Y 282.149,Z 717.465,A -85,B 0,C 180,E1 16130.456,E2 16130.456} C_VEL
LIN {X 0,Y 288.209,Z 698.137,A -85,B 0,C 180,E1 16136.912,E2 16136.912} C_VEL
LIN {X 0,Y 297.494,Z 672.951,A -85,B 0,C 180,E1 16142.601,E2 16142.601} C_VEL
LIN {X 0,Y 307.977,Z 645.153,A -85,B 0,C 180,E1 16146.818,E2 16146.818} C_VEL
LIN {X 0,Y 318.449,Z 613.978,A -85,B 0,C 180,E1 16149.972,E2 16149.972} C_VEL
LIN {X 0,Y 321.345,Z 603.364,A -85,B 0,C 180,E1 16150.841,E2 16150.841} C_VEL
LIN {X 0,Y 318.953,Z 591.302,A -85,B 0,C 180,E1 16153.731,E2 16153.731} C_VEL
LIN {X 0,Y 316.434,Z 584.253,A -85,B 0,C 180,E1 16156.735,E2 16156.735} C_VEL
LIN {X 0,Y 314.537,Z 581.283,A -85,B 0,C 180,E1 16161.274,E2 16161.274} C_VEL
LIN {X 0,Y 314.747,Z 585.781,A -85,B 0,C 180,E1 16165.488,E2 16165.488} C_VEL
LIN {X 0,Y 315.415,Z 595.645,A -85,B 0,C 180,E1 16169.24,E2 16169.24} C_VEL
LIN {X 0,Y 315.39,Z 597.913,A -85,B 0,C 180,E1 16169.869,E2 16169.869} C_VEL
LIN {X 0,Y 313.187,Z 604.499,A -85,B 0,C 180,E1 16170.797,E2 16170.797} C_VEL
LIN {X 0,Y 306.435,Z 616.855,A -85,B 0,C 180,E1 16171.91,E2 16171.91} C_VEL
LIN {X 0,Y 296.318,Z 638.387,A -85,B 0,C 180,E1 16176.284,E2 16176.284} C_VEL
LIN {X 0,Y 288.23,Z 652.784,A -85,B 0,C 180,E1 16180.845,E2 16180.845} C_VEL
LIN {X 0,Y 281.743,Z 662.283,A -85,B 0,C 180,E1 16186.016,E2 16186.016} C_VEL
LIN {X 0,Y 277.647,Z 666.057,A -85,B 0,C 180,E1 16190.595,E2 16190.595} C_VEL
LIN {X 0,Y 275.841,Z 666.349,A -85,B 0,C 180,E1 16193.708,E2 16193.708} C_VEL
LIN {X 0,Y 273.937,Z 663.562,A -85,B 0,C 180,E1 16198.426,E2 16198.426} C_VEL
LIN {X 0,Y 273.199,Z 654.355,A -85,B 0,C 180,E1 16204.299,E2 16204.299} C_VEL
LIN {X 0,Y 273.795,Z 639.876,A -85,B 0,C 180,E1 16209.559,E2 16209.559} C_VEL
LIN {X 0,Y 275.472,Z 619.995,A -85,B 0,C 180,E1 16214.329,E2 16214.329} C_VEL
LIN {X 0,Y 277.815,Z 594.894,A -85,B 0,C 180,E1 16218.398,E2 16218.398} C_VEL
LIN {X 0,Y 278.657,Z 575.494,A -85,B 0,C 180,E1 16220.667,E2 16220.667} C_VEL
LIN {X 0,Y 272.736,Z 545.145,A -85,B 0,C 180,E1 16223.45,E2 16223.45} C_VEL
LIN {X 0,Y 268.535,Z 526.81,A -85,B 0,C 180,E1 16224.684,E2 16224.684} C_VEL
LIN {X 0,Y 267.844,Z 526.81,A -85,B 0,C 180,E1 16234.432,E2 16234.432} C_VEL
LIN {X 0,Y 267.662,Z 526.81,A -85,B 0,C 180,E1 16242.76,E2 16242.76} C_VEL
LIN {X 0,Y 267.781,Z 526.81,A -85,B 0,C 180,E1 16251.531,E2 16251.531} C_VEL
LIN {X 0,Y 268.012,Z 526.81,A -85,B 0,C 180,E1 16259.432,E2 16259.432} C_VEL
LIN {X 0,Y 268.4,Z 526.81,A -85,B 0,C 180,E1 16266.733,E2 16266.733} C_VEL
LIN {X 0,Y 268.83,Z 526.81,A -85,B 0,C 180,E1 16273.636,E2 16273.636} C_VEL
LIN {X 0,Y 269.322,Z 526.81,A -85,B 0,C 180,E1 16280.283,E2 16280.283} C_VEL
LIN {X 0,Y 270.024,Z 526.81,A -85,B 0,C 180,E1 16286.778,E2 16286.778} C_VEL
LIN {X 0,Y 270.014,Z 526.81,A -85,B 0,C 180,E1 16293.207,E2 16293.207} C_VEL
LIN {X 0,Y 269.382,Z 526.81,A -85,B 0,C 180,E1 16299.7,E2 16299.7} C_VEL
LIN {X 0,Y 268.83,Z 526.81,A -85,B 0,C 180,E1 16306.749,E2 16306.749} C_VEL
LIN {X 0,Y 268.267,Z 526.81,A -85,B 0,C 180,E1 16315.425,E2 16315.425} C_VEL
LIN {X 0,Y 267.838,Z 526.81,A -85,B 0,C 180,E1 16324.413,E2 16324.413} C_VEL
LIN {X 0,Y 267.649,Z 526.81,A -85,B 0,C 180,E1 16332.742,E2 16332.742} C_VEL
LIN {X 0,Y 267.747,Z 526.81,A -85,B 0,C 180,E1 16341.525,E2 16341.525} C_VEL
LIN {X 0,Y 267.977,Z 526.81,A -85,B 0,C 180,E1 16349.426,E2 16349.426} C_VEL
LIN {X 0,Y 268.366,Z 526.81,A -85,B 0,C 180,E1 16356.729,E2 16356.729} C_VEL
LIN {X 0,Y 268.848,Z 526.81,A -85,B 0,C 180,E1 16363.636,E2 16363.636} C_VEL
LIN {X 0,Y 269.361,Z 526.81,A -85,B 0,C 180,E1 16371.804,E2 16371.804} C_VEL
LIN {X 0,Y 270.285,Z 526.81,A -85,B 0,C 180,E1 16379.99,E2 16379.99} C_VEL
LIN {X 0,Y 269.619,Z 526.81,A -85,B 0,C 180,E1 16386.438,E2 16386.438} C_VEL
LIN {X 0,Y 269.074,Z 526.81,A -85,B 0,C 180,E1 16392.997,E2 16392.997} C_VEL
LIN {X 0,Y 268.634,Z 526.81,A -85,B 0,C 180,E1 16399.754,E2 16399.754} C_VEL
LIN {X 0,Y 268.218,Z 526.81,A -85,B 0,C 180,E1 16406.833,E2 16406.833} C_VEL
LIN {X 0,Y 267.867,Z 526.81,A -85,B 0,C 180,E1 16414.404,E2 16414.404} C_VEL
LIN {X 0,Y 267.588,Z 526.81,A -85,B 0,C 180,E1 16422.748,E2 16422.748} C_VEL
LIN {X 0,Y 268.024,Z 527.299,A -85,B 0,C 180,E1 16432.04,E2 16432.04} C_VEL
LIN {X 0,Y 287.013,Z 591.706,A -85,B 0,C 180,E1 16435.78,E2 16435.78} C_VEL
LIN {X 0,Y 287.815,Z 601.683,A -85,B 0,C 180,E1 16436.432,E2 16436.432} C_VEL
LIN {X 0,Y 283.726,Z 634.646,A -85,B 0,C 180,E1 16439.118,E2 16439.118} C_VEL
LIN {X 0,Y 279.329,Z 663.53,A -85,B 0,C 180,E1 16442.768,E2 16442.768} C_VEL
LIN {X 0,Y 275.656,Z 688.752,A -85,B 0,C 180,E1 16447.397,E2 16447.397} C_VEL
LIN {X 0,Y 273.183,Z 710.265,A -85,B 0,C 180,E1 16453.092,E2 16453.092} C_VEL
LIN {X 0,Y 272.545,Z 724.893,A -85,B 0,C 180,E1 16458.796,E2 16458.796} C_VEL
LIN {X 0,Y 272.962,Z 734.066,A -85,B 0,C 180,E1 16464.517,E2 16464.517} C_VEL
LIN {X 0,Y 273.295,Z 738.192,A -85,B 0,C 180,E1 16470.008,E2 16470.008} C_VEL
LIN {X 0,Y 272.265,Z 737.458,A -85,B 0,C 180,E1 16476.393,E2 16476.393} C_VEL
LIN {X 0,Y 271.853,Z 730.684,A -85,B 0,C 180,E1 16483.456,E2 16483.456} C_VEL
LIN {X 0,Y 274.225,Z 718.157,A -85,B 0,C 180,E1 16490.487,E2 16490.487} C_VEL
LIN {X 0,Y 280.702,Z 699.175,A -85,B 0,C 180,E1 16497.354,E2 16497.354} C_VEL
LIN {X 0,Y 290.388,Z 675.12,A -85,B 0,C 180,E1 16503.189,E2 16503.189} C_VEL
LIN {X 0,Y 301.88,Z 647.338,A -85,B 0,C 180,E1 16507.689,E2 16507.689} C_VEL
LIN {X 0,Y 313.425,Z 616.285,A -85,B 0,C 180,E1 16511.013,E2 16511.013} C_VEL
LIN {X 0,Y 316.423,Z 606.795,A -85,B 0,C 180,E1 16511.825,E2 16511.825} C_VEL
LIN {X 0,Y 314.7,Z 596.593,A -85,B 0,C 180,E1 16514.578,E2 16514.578} C_VEL
LIN {X 0,Y 312.791,Z 590.873,A -85,B 0,C 180,E1 16517.352,E2 16517.352} C_VEL
LIN {X 0,Y 311.377,Z 588.474,A -85,B 0,C 180,E1 16521.088,E2 16521.088} C_VEL
LIN {X 0,Y 311.019,Z 592.244,A -85,B 0,C 180,E1 16525.015,E2 16525.015} C_VEL
LIN {X 0,Y 310.877,Z 600.605,A -85,B 0,C 180,E1 16528.467,E2 16528.467} C_VEL
LIN {X 0,Y 309.199,Z 610.323,A -85,B 0,C 180,E1 16530.893,E2 16530.893} C_VEL
LIN {X 0,Y 306.435,Z 616.855,A -85,B 0,C 180,E1 16531.91,E2 16531.91} C_VEL
LIN {X 0,Y 298.423,Z 630.002,A -85,B 0,C 180,E1 16533.557,E2 16533.557} C_VEL
LIN {X 0,Y 291.025,Z 640.281,A -85,B 0,C 180,E1 16535.187,E2 16535.187} C_VEL
LIN {X 0,Y 290.254,Z 641.518,A -85,B 0,C 180,E1 16535.5,E2 16535.5} C_VEL
LIN {X 0,Y 281.282,Z 655.782,A -85,B 0,C 180,E1 16540.352,E2 16540.352} C_VEL
LIN {X 0,Y 274.056,Z 664.845,A -85,B 0,C 180,E1 16545.97,E2 16545.97} C_VEL
LIN {X 0,Y 270.037,Z 667.745,A -85,B 0,C 180,E1 16550.327,E2 16550.327} C_VEL
LIN {X 0,Y 268.117,Z 667.763,A -85,B 0,C 180,E1 16553.526,E2 16553.526} C_VEL
LIN {X 0,Y 266.117,Z 664.484,A -85,B 0,C 180,E1 16558.38,E2 16558.38} C_VEL
LIN {X 0,Y 265.323,Z 654.75,A -85,B 0,C 180,E1 16564.427,E2 16564.427} C_VEL
LIN {X 0,Y 265.964,Z 639.722,A -85,B 0,C 180,E1 16569.843,E2 16569.843} C_VEL
LIN {X 0,Y 267.75,Z 619.138,A -85,B 0,C 180,E1 16574.751,E2 16574.751} C_VEL
LIN {X 0,Y 270.139,Z 594.134,A -85,B 0,C 180,E1 16578.817,E2 16578.817} C_VEL
LIN {X 0,Y 270.893,Z 576.611,A -85,B 0,C 180,E1 16580.904,E2 16580.904} C_VEL
LIN {X 0,Y 265.111,Z 546.686,A -85,B 0,C 180,E1 16583.757,E2 16583.757} C_VEL
LIN {X 0,Y 260.54,Z 526.81,A -85,B 0,C 180,E1 16585.261,E2 16585.261} C_VEL
LIN {X 0,Y 259.979,Z 526.81,A -85,B 0,C 180,E1 16591.621,E2 16591.621} C_VEL
LIN {X 0,Y 259.657,Z 526.81,A -85,B 0,C 180,E1 16599.908,E2 16599.908} C_VEL
LIN {X 0,Y 259.658,Z 526.81,A -85,B 0,C 180,E1 16609.303,E2 16609.303} C_VEL
LIN {X 0,Y 259.877,Z 526.81,A -85,B 0,C 180,E1 16614.666,E2 16614.666} C_VEL
LIN {X 0,Y 260.198,Z 526.81,A -85,B 0,C 180,E1 16622.248,E2 16622.248} C_VEL
LIN {X 0,Y 260.616,Z 526.81,A -85,B 0,C 180,E1 16629.591,E2 16629.591} C_VEL
LIN {X 0,Y 261.07,Z 526.81,A -85,B 0,C 180,E1 16636.578,E2 16636.578} C_VEL
LIN {X 0,Y 261.666,Z 526.81,A -85,B 0,C 180,E1 16643.347,E2 16643.347} C_VEL
LIN {X 0,Y 262.407,Z 526.81,A -85,B 0,C 180,E1 16649.992,E2 16649.992} C_VEL
LIN {X 0,Y 261.715,Z 526.81,A -85,B 0,C 180,E1 16656.636,E2 16656.636} C_VEL
LIN {X 0,Y 261.16,Z 526.81,A -85,B 0,C 180,E1 16663.401,E2 16663.401} C_VEL
LIN {X 0,Y 260.498,Z 526.81,A -85,B 0,C 180,E1 16671.552,E2 16671.552} C_VEL
LIN {X 0,Y 260.062,Z 526.81,A -85,B 0,C 180,E1 16679.141,E2 16679.141} C_VEL
LIN {X 0,Y 259.817,Z 526.81,A -85,B 0,C 180,E1 16685.634,E2 16685.634} C_VEL
LIN {X 0,Y 259.559,Z 526.81,A -85,B 0,C 180,E1 16694.415,E2 16694.415} C_VEL
LIN {X 0,Y 259.653,Z 526.81,A -85,B 0,C 180,E1 16700.091,E2 16700.091} C_VEL
LIN {X 0,Y 259.989,Z 526.81,A -85,B 0,C 180,E1 16708.381,E2 16708.381} C_VEL
LIN {X 0,Y 260.384,Z 526.81,A -85,B 0,C 180,E1 16715.972,E2 16715.972} C_VEL
LIN {X 0,Y 260.875,Z 526.81,A -85,B 0,C 180,E1 16723.121,E2 16723.121} C_VEL
LIN {X 0,Y 261.435,Z 526.81,A -85,B 0,C 180,E1 16731.841,E2 16731.841} C_VEL
LIN {X 0,Y 262.377,Z 526.81,A -85,B 0,C 180,E1 16739.99,E2 16739.99} C_VEL
LIN {X 0,Y 261.67,Z 526.81,A -85,B 0,C 180,E1 16746.635,E2 16746.635} C_VEL
LIN {X 0,Y 261.105,Z 526.81,A -85,B 0,C 180,E1 16753.401,E2 16753.401} C_VEL
LIN {X 0,Y 260.473,Z 526.81,A -85,B 0,C 180,E1 16761.58,E2 16761.58} C_VEL
LIN {X 0,Y 260.065,Z 526.81,A -85,B 0,C 180,E1 16769.174,E2 16769.174} C_VEL
LIN {X 0,Y 259.831,Z 526.81,A -85,B 0,C 180,E1 16775.627,E2 16775.627} C_VEL
LIN {X 0,Y 259.493,Z 526.81,A -85,B 0,C 180,E1 16784.423,E2 16784.423} C_VEL
LIN {X 0,Y 260.017,Z 527.125,A -85,B 0,C 180,E1 16791.479,E2 16791.479} C_VEL
LIN {X 0,Y 278.888,Z 591.505,A -85,B 0,C 180,E1 16795.348,E2 16795.348} C_VEL
LIN {X 0,Y 280.23,Z 601.038,A -85,B 0,C 180,E1 16796.021,E2 16796.021} C_VEL
LIN {X 0,Y 276.135,Z 633.234,A -85,B 0,C 180,E1 16798.708,E2 16798.708} C_VEL
LIN {X 0,Y 271.47,Z 663.29,A -85,B 0,C 180,E1 16802.613,E2 16802.613} C_VEL
LIN {X 0,Y 267.599,Z 689.33,A -85,B 0,C 180,E1 16807.609,E2 16807.609} C_VEL
LIN {X 0,Y 265.279,Z 710.182,A -85,B 0,C 180,E1 16813.427,E2 16813.427} C_VEL
LIN {X 0,Y 264.77,Z 724.398,A -85,B 0,C 180,E1 16819.297,E2 16819.297} C_VEL
LIN {X 0,Y 265.266,Z 733.136,A -85,B 0,C 180,E1 16825.096,E2 16825.096} C_VEL
LIN {X 0,Y 265.538,Z 736.685,A -85,B 0,C 180,E1 16830.008,E2 16830.008} C_VEL
LIN {X 0,Y 264.389,Z 736.179,A -85,B 0,C 180,E1 16836.585,E2 16836.585} C_VEL
LIN {X 0,Y 264.049,Z 729.398,A -85,B 0,C 180,E1 16844.113,E2 16844.113} C_VEL
LIN {X 0,Y 266.974,Z 716.468,A -85,B 0,C 180,E1 16851.639,E2 16851.639} C_VEL
LIN {X 0,Y 274.361,Z 697.594,A -85,B 0,C 180,E1 16858.638,E2 16858.638} C_VEL
LIN {X 0,Y 285.054,Z 673.486,A -85,B 0,C 180,E1 16864.602,E2 16864.602} C_VEL
LIN {X 0,Y 297.88,Z 645.05,A -85,B 0,C 180,E1 16869.22,E2 16869.22} C_VEL
LIN {X 0,Y 310.543,Z 613.486,A -85,B 0,C 180,E1 16872.55,E2 16872.55} C_VEL
LIN {X 0,Y 311.49,Z 608.825,A -85,B 0,C 180,E1 16873.204,E2 16873.204} C_VEL
LIN {X 0,Y 310.16,Z 600.777,A -85,B 0,C 180,E1 16875.903,E2 16875.903} C_VEL
LIN {X 0,Y 308.747,Z 596.957,A -85,B 0,C 180,E1 16878.468,E2 16878.468} C_VEL
LIN {X 0,Y 307.568,Z 596.214,A -85,B 0,C 180,E1 16881.976,E2 16881.976} C_VEL
LIN {X 0,Y 307.006,Z 600.132,A -85,B 0,C 180,E1 16885.365,E2 16885.365} C_VEL
LIN {X 0,Y 305.936,Z 608.5,A -85,B 0,C 180,E1 16888.607,E2 16888.607} C_VEL
LIN {X 0,Y 303.818,Z 615.202,A -85,B 0,C 180,E1 16890.121,E2 16890.121} C_VEL
LIN {X 0,Y 292.767,Z 637.034,A -85,B 0,C 180,E1 16894.346,E2 16894.346} C_VEL
LIN {X 0,Y 290.254,Z 641.518,A -85,B 0,C 180,E1 16895.5,E2 16895.5} C_VEL
LIN {X 0,Y 281.687,Z 651.761,A -85,B 0,C 180,E1 16897.819,E2 16897.819} C_VEL
LIN {X 0,Y 274.074,Z 659.159,A -85,B 0,C 180,E1 16900.066,E2 16900.066} C_VEL
LIN {X 0,Y 273.369,Z 659.975,A -85,B 0,C 180,E1 16900.458,E2 16900.458} C_VEL
LIN {X 0,Y 267.087,Z 666.681,A -85,B 0,C 180,E1 16905.232,E2 16905.232} C_VEL
LIN {X 0,Y 262.444,Z 669.442,A -85,B 0,C 180,E1 16910.044,E2 16910.044} C_VEL
LIN {X 0,Y 259.558,Z 668.272,A -85,B 0,C 180,E1 16914.991,E2 16914.991} C_VEL
LIN {X 0,Y 257.588,Z 661.341,A -85,B 0,C 180,E1 16921.288,E2 16921.288} C_VEL
LIN {X 0,Y 257.6,Z 648.559,A -85,B 0,C 180,E1 16927.185,E2 16927.185} C_VEL
LIN {X 0,Y 258.773,Z 631.624,A -85,B 0,C 180,E1 16932.255,E2 16932.255} C_VEL
LIN {X 0,Y 261.073,Z 607.819,A -85,B 0,C 180,E1 16937.071,E2 16937.071} C_VEL
LIN {X 0,Y 263.56,Z 580.244,A -85,B 0,C 180,E1 16940.837,E2 16940.837} C_VEL
LIN {X 0,Y 257.838,Z 550.048,A -85,B 0,C 180,E1 16943.896,E2 16943.896} C_VEL
LIN {X 0,Y 252.576,Z 526.81,A -85,B 0,C 180,E1 16945.653,E2 16945.653} C_VEL
LIN {X 0,Y 251.948,Z 526.81,A -85,B 0,C 180,E1 16952.752,E2 16952.752} C_VEL
LIN {X 0,Y 251.633,Z 526.81,A -85,B 0,C 180,E1 16961.454,E2 16961.454} C_VEL
LIN {X 0,Y 251.66,Z 526.81,A -85,B 0,C 180,E1 16968.552,E2 16968.552} C_VEL
LIN {X 0,Y 251.967,Z 526.81,A -85,B 0,C 180,E1 16977.288,E2 16977.288} C_VEL
LIN {X 0,Y 252.375,Z 526.81,A -85,B 0,C 180,E1 16985.16,E2 16985.16} C_VEL
LIN {X 0,Y 252.95,Z 526.81,A -85,B 0,C 180,E1 16993.303,E2 16993.303} C_VEL
LIN {X 0,Y 253.728,Z 526.81,A -85,B 0,C 180,E1 17003.138,E2 17003.138} C_VEL
LIN {X 0,Y 254.505,Z 526.81,A -85,B 0,C 180,E1 17009.992,E2 17009.992} C_VEL
LIN {X 0,Y 253.796,Z 526.81,A -85,B 0,C 180,E1 17016.844,E2 17016.844} C_VEL
LIN {X 0,Y 253.173,Z 526.81,A -85,B 0,C 180,E1 17023.832,E2 17023.832} C_VEL
LIN {X 0,Y 252.646,Z 526.81,A -85,B 0,C 180,E1 17031.065,E2 17031.065} C_VEL
LIN {X 0,Y 252.195,Z 526.81,A -85,B 0,C 180,E1 17038.695,E2 17038.695} C_VEL
LIN {X 0,Y 251.707,Z 526.81,A -85,B 0,C 180,E1 17046.969,E2 17046.969} C_VEL
LIN {X 0,Y 251.611,Z 526.81,A -85,B 0,C 180,E1 17056.216,E2 17056.216} C_VEL
LIN {X 0,Y 251.731,Z 526.81,A -85,B 0,C 180,E1 17063.014,E2 17063.014} C_VEL
LIN {X 0,Y 252.198,Z 526.81,A -85,B 0,C 180,E1 17071.286,E2 17071.286} C_VEL
LIN {X 0,Y 252.617,Z 526.81,A -85,B 0,C 180,E1 17078.913,E2 17078.913} C_VEL
